	(* 4=zur *)							
	IF hm_zur
		AND NOT temp_end_zur
		AND NOT temp_stoer_zur
		AND NOT temp_stoer_vor_zur
	THEN
		inout_visu.status:=4;									
	END_IF									
	(* 5=ist zur *)							
	IF (temp_end_zur
		OR (NOT inout_visu.para.ueberwachung_zur_aktiv
				AND hm_zur))
		AND NOT temp_end_vor
		AND NOT temp_stoer_zur
		AND NOT temp_stoer_vor_zur
	THEN
		inout_visu.status:=5;									
	END_IF															
	(* 6=Fehler zurück *)								
	IF temp_stoer_zur
	THEN
		inout_visu.status:=6;
	END_IF
	(* 7=Fehler vor zur	*)
	IF temp_stoer_vor_zur
	THEN
		inout_visu.status:=7;
	END_IF

	
(***** Endlagen direkt an die Visu weiter reichen ***********************************************************************************************************)
	out_vor_visu:=in_endlage_vor;
	out_zur_visu:=in_endlage_zur;


(***** IN Start-Befehle Hand und Automatik löschen **********************************************************************************************************)
	inout_ansteuerung.in_auto_vor:=FALSE;
	inout_ansteuerung.in_auto_zur:=FALSE;
	inout_ansteuerung.in_aus := FALSE;
	inout_visu.hand_vor:=FALSE;
	inout_visu.hand_zur:=FALSE;
	hm_timer_reset:=TRUE;

METHOD M_AutoVor : BOOL
VAR_INPUT
	Active		: BOOL;
END_VAR
inout_ansteuerung.in_auto_vor := Active;
IF inout_ansteuerung.out_ist_vor OR NOT Active THEN
	M_AutoVor := TRUE;
END_IF
END_METHOD

METHOD M_AutoZur : BOOL
VAR_INPUT
	Active		: BOOL;
END_VAR
inout_ansteuerung.in_auto_zur := Active;
IF inout_ansteuerung.out_ist_zur OR NOT Active THEN
	M_AutoZur := TRUE;
END_IF
END_METHOD

END_FUNCTION_BLOCK

// ---- 3400_Bohraggregat/Hardware_3400.TcPOU

PROGRAM Hardware_3400
VAR
    // Servos *********************************************************************
	fbX_Achse										: FB_Achse_NC_PTP_Beckhoff; 
	fbY_Achse										: FB_Achse_NC_PTP_Beckhoff; 

    // Frequenzumrichter **********************************************************
	fbBohraggr_Schluessel_ob						: FB_SEW_MOVITRAC_C_CoE;

    // Sensorik *******************************************************************
    fbStillBohraggr_Schluessel_ob          			: FB_Belegt;

    // Ventile ********************************************************************
    fbSchluessel_ob_Bohrhub                			: FB_Ventil_V2;

    // ***** Hilfsmerker***********************************************************
    (*
        Ventile sind über den DUT_Ventil_para vorparametriert
                ueberwachung_vor_aktiv    : BOOL := TRUE;   // 0 = Endlagenüberwachung vor deaktiviert
                ueberwachung_zur_aktiv    : BOOL := TRUE;   // 0 = Endlagenüberwachung zurück deaktiviert
                ausgang_vor_halten        : BOOL := FALSE;  // 1 = Ausgang immer Ein, sonst 0 in Endlage/1 nicht in Endlage
                ausgang_zur_halten        : BOOL := FALSE;  // 1 = Ausgang immer Ein, sonst 0 in Endlage/1 nicht in Endlage
                entprellen_vor_aktiv      : BOOL := TRUE;   // 0 = Endlage sofort überwachen wenn einmal erreicht
                entprellen_zur_aktiv      : BOOL := TRUE;   // 0 = Endlage sofort überwachen wenn einmal erreicht
                ueberwachungszeit_vor     : TIME := T#10S;  // Überwachungszeit in ms (0-30000ms)
                ueberwachungszeit_zur     : TIME := T#10S;  // Überwachungszeit in ms (0-30000ms)
                entprellungszeit_vor      : TIME := T#50MS; // Entprellungszeit in ms (0-10000ms)
                entprellungszeit_zur      : TIME := T#50MS; // Entprellungszeit in ms (0-10000ms)

        falls etwas anderes gewünscht ist, kann man gezielt für das Ventil die Parameter anpassen
        Beispiel:   ***.para.ausgang_vor_halten := TRUE;
                    ***.para.entprellungszeit_vor := T#100MS;
    *)
END_VAR


// Aktionen aufrufen
//_________________________________________________
	A_Sensorik();
	A_Umrichter();
	A_Ventile();
	A_Servo();

ACTION A_Sensorik:
					
// ***** Sensorik entprellen *********************************************************
	//********************************************************************************
fbStillBohraggr_Schluessel_ob	(	in_Sensor:=,
									in_zeit_aus:=T#100MS,
									in_zeit_aus:=T#100MS,
									Q=>);
END_ACTION

ACTION A_Servo:
					
// ***** Servoregler *****************************************************************
	//********************************************************************************
	GVL_3400.X_Achse_steuern.Reglersperre	:= FALSE;
	GVL_3400.X_Achse_steuern.Freigabe 		:= FALSE;
	
	fbX_Achse(
	in_Reglersperre				:= GVL_3400.X_Achse_steuern.Reglersperre, 
	in_Freigabe					:= GVL_3400.X_Achse_steuern.Freigabe,
	in_Reset					:= GVL_Visu_3400.SteuerStatus.reset   
								OR GVL_0000.stoerung_quitt,                      
	in_Hand						:= GVL_Visu_3400.SteuerStatus.hand,              
	in_Auto						:= GVL_Visu_3400.SteuerStatus.auto,                 
	in_Auto_Override			:= GVL_Visu_0000.override,    
	in_Auto_pos					:= , 
	in_PosFenster				:= 0.05, 
	in_Ref_pos					:= 0.0, 
	in_HomingOption				:= , 
	in_EndlageRef				:= , 
	in_DirRef					:= , 
	in_PosEa					:= ,                                       
	out_ist_pos					=> GVL_3400.X_Achse_status.ist_pos, 
	out_in_pos					=> GVL_3400.X_Achse_status.in_pos,   
	out_ziel_pos				=> GVL_3400.X_Achse_status.ziel_pos, 
	out_nicht_ref				=> GVL_3400.X_Achse_status.nicht_ref,      
	out_bremse					=> GVL_3400.X_Achse_status.bremse,           
	out_Achs_Status				=> GVL_3400.X_Achse_status.Achs_Status,  
	inout_NC					:= EAs_3400.ea_X_Achse, 
	inout_service				:= GVL_Visu_3400.X_Achse, 
	inout_Ref_start				:= GVL_3400.X_Achse_steuern.Ref_start, 
	inout_Auto_start			:= GVL_3400.X_Achse_steuern.Auto_start, 
	inout_Auto_stop				:= GVL_3400.X_Achse_steuern.Auto_stop);
	
	GVL_Meldungen.Diagnose_3000.Nr_034	:= fbX_Achse.out_Achs_ErrorID;	
	GVL_Meldungen.Meldungen_3000.Nr_034 := fbX_Achse.out_Achs_Error OR fbX_Achse.out_FB_Error OR fbX_Achse.out_Achs_ErrorID <> 0;		
	GVL_Meldungen.Meldungen_3000.Nr_035 := FALSE;
	GVL_Meldungen.Meldungen_3000.Nr_036 := FALSE;
	//********************************************************************************
					
					
	GVL_3400.Y_Achse_steuern.Reglersperre	:= FALSE;
	GVL_3400.Y_Achse_steuern.Freigabe 		:= FALSE;
	
	fbY_Achse(
	in_Reglersperre				:= GVL_3400.Y_Achse_steuern.Reglersperre, 
	in_Freigabe					:= GVL_3400.Y_Achse_steuern.Freigabe,
	in_Reset					:= GVL_Visu_3400.SteuerStatus.reset   
								OR GVL_0000.stoerung_quitt,                      
	in_Hand						:= GVL_Visu_3400.SteuerStatus.hand,              
	in_Auto						:= GVL_Visu_3400.SteuerStatus.auto,                 
	in_Auto_Override			:= GVL_Visu_0000.override,    
	in_Auto_pos					:= , 
	in_PosFenster				:= 0.05, 
	in_Ref_pos					:= 0.0, 
	in_HomingOption				:= , 
	in_EndlageRef				:= , 
	in_DirRef					:= , 
	in_PosEa					:= ,                                       
	out_ist_pos					=> GVL_3400.Y_Achse_status.ist_pos, 
	out_in_pos					=> GVL_3400.Y_Achse_status.in_pos,   
	out_ziel_pos				=> GVL_3400.Y_Achse_status.ziel_pos, 
	out_nicht_ref				=> GVL_3400.Y_Achse_status.nicht_ref,      
	out_bremse					=> GVL_3400.Y_Achse_status.bremse,           
	out_Achs_Status				=> GVL_3400.Y_Achse_status.Achs_Status,  
	inout_NC					:= EAs_3400.ea_Y_Achse, 
	inout_service				:= GVL_Visu_3400.Y_Achse, 
	inout_Ref_start				:= GVL_3400.Y_Achse_steuern.Ref_start, 
	inout_Auto_start			:= GVL_3400.Y_Achse_steuern.Auto_start, 
	inout_Auto_stop				:= GVL_3400.Y_Achse_steuern.Auto_stop);
	
	GVL_Meldungen.Diagnose_3000.Nr_037	:= fbY_Achse.out_Achs_ErrorID;	
	GVL_Meldungen.Meldungen_3000.Nr_037 := fbY_Achse.out_Achs_Error OR fbY_Achse.out_FB_Error OR fbY_Achse.out_Achs_ErrorID <> 0;		
	GVL_Meldungen.Meldungen_3000.Nr_038 := FALSE;
	GVL_Meldungen.Meldungen_3000.Nr_039 := FALSE;
END_ACTION

ACTION A_Umrichter:
	
// ***** Frequenzumrichter ******************************************************
// ******************************************************************************
				
	GVL_Visu_3400.Bohraggr_Schluessel_ob	.Para.Speed_Hand		:= 0;
	GVL_Visu_3400.Bohraggr_Schluessel_ob	.Para.Beschleunigung 	:= 0;
	GVL_Visu_3400.Bohraggr_Schluessel_ob	.Para.Verzoegerung 		:= 0;
	GVL_Visu_3400.Bohraggr_Schluessel_ob	.Para.Einheit			:= 1;

	fbBohraggr_Schluessel_ob	(	PD_IN	:=EAs_3400.e_Bohraggr_Schluessel_ob	,
			IN_ReglerSperre			:=,
			IN_SteuerStatus			:=GVL_Visu_3400.SteuerStatus,
			IN_Ethercat_Adresse		:=,
			IN_Ethercat_Name		:='',
			IN_QUITTIEREN			:= GVL_0000.stoerung_quitt,
			IN_OVERRIDE				:= GVL_Visu_0000.override,
			PD_OUT					=> EAs_3400.a_Bohraggr_Schluessel_ob	,
			OUT_Stoerung			=> GVL_Meldungen.Meldungen_3000.Nr_007,
			OUT_Fehlernummer		=> GVL_Meldungen.Diagnose_3000.Nr_007,
			OUT_Status				=> GVL_3400.Bohraggr_Schluessel_ob_status,
			inout_visu				:= GVL_Visu_3400.Bohraggr_Schluessel_ob	,
			inout_steuern			:= GVL_3400.Bohraggr_Schluessel_ob_steuern);
	
			GVL_3400.Bohraggr_Schluessel_ob_steuern.vor := FALSE;
			GVL_3400.Bohraggr_Schluessel_ob_steuern.zur := FALSE;
			GVL_3400.Bohraggr_Schluessel_ob_steuern.speed := 0;
END_ACTION

ACTION A_Ventile:
	
// ***** Ventile *********************************************************************
	//********************************************************************************	
	
	GVL_Visu_3400.Schluessel_ob_Bohrhub.para.ausgang_vor_halten:=TRUE;	
	GVL_Visu_3400.Schluessel_ob_Bohrhub.para.ausgang_zur_halten:=TRUE;	
	GVL_Visu_3400.Schluessel_ob_Bohrhub.para.ueberwachung_vor_aktiv:=TRUE;	
	GVL_Visu_3400.Schluessel_ob_Bohrhub.para.ueberwachung_zur_aktiv:=TRUE;	
	GVL_Visu_3400.Schluessel_ob_Bohrhub.para.entprellungszeit_vor:=T#50S;	
	GVL_Visu_3400.Schluessel_ob_Bohrhub.para.entprellungszeit_zur:=T#50MS;	
	fbSchluessel_ob_Bohrhub (	in_endlage_vor:= EAs_3400.e_FR_3400_Druecker_Schluesselloch_oben_Bohraggregat_7_Bohrhub_ist_oben,
								in_endlage_zur:= EAs_3400.e_FR_3400_Druecker_Schluesselloch_oben_Bohraggregat_7_Bohrhub_ist_unten,
								in_hand:=GVL_Visu_3400.SteuerStatus.hand,
								in_auto:=GVL_Visu_3400.SteuerStatus.auto,
								in_quit:=GVL_Visu_3400.SteuerStatus.reset 
								OR GVL_0000.stoerung_quitt,
								out_vor=>EAs_3400.a_FR_3400_Druecker_Schluesselloch_oben_Bohraggregat_7_Bohrhub_heben,
								out_zur=>EAs_3400.a_FR_3400_Druecker_Schluesselloch_oben_Bohraggregat_7_Bohrhub_senken,
								out_stoerung_vor=> GVL_Meldungen.Meldungen_3000.Nr_070,
								out_stoerung_zur=> GVL_Meldungen.Meldungen_3000.Nr_071,
								out_stoerung_vorzur=> GVL_Meldungen.Meldungen_3000.Nr_072,
								inout_ansteuerung:=GVL_3400.Schluessel_ob_Bohrhub ,
								inout_visu:=GVL_Visu_3400.Schluessel_ob_Bohrhub );
END_ACTION

END_PROGRAM

// ---- 3510_Transport/Ablauf_3510.TcPOU

PROGRAM Ablauf_3510
VAR
    // TODO: lokale Variablen fuer den Ablauf deklarieren
END_VAR


// TODO: Hauptprogramm-Code fuer Ablauf hier einfuegen


METHOD M_VisuKomm : BOOL
VAR_INPUT
    Nr          : INT;
END_VAR
VAR_IN_OUT
    anVisu      : INT;
    vonVisu     : INT;
END_VAR

VAR_INST
    result                  : INT;
    ton_DatenUngueltig      : TON;
    ton_DatenTimeout        : TON;
    sc                      : INT;
END_VAR

// Schnistelle zur VISU Kommunikation
// Starttrigger belegen als Antwort wird auf die 5= gut oder 9=schlecht gewartet.
// Kommunikationstimeout nach 5 Sekunden und wird automatisch wieder neugestartet

ton_DatenTimeout(IN:= anVisu <> 0 AND vonVisu = 0, PT:=T#3S);
ton_DatenUngueltig(IN:= sc = 20, PT:=T#500MS);

CASE sc OF
    0:  // Anfrage starten und auf Antwort warten
        anVisu := Nr;
        result := 0;
        IF vonVisu <> 0 THEN
            IF (vonVisu MOD Nr) = 5 THEN
                sc := 10;
            ELSIF (vonVisu MOD Nr) = 9 THEN
                sc := 20;
            END_IF
        ELSIF ton_DatenTimeout.Q THEN
            sc := 20;
        END_IF

    10: // Antwort 5 erhalten
        anVisu := 0;
        IF vonVisu = 0 THEN
            M_VisuKomm := TRUE;
            result := 1;
            sc := 0;
        END_IF

    20: // Timeout, 1 Sekunde warten und erneut antriggern
        IF ton_DatenUngueltig.Q THEN
            anVisu := 0;
            IF vonVisu = 0 THEN
                result := -1;
                sc := 0;
            END_IF
        END_IF

END_CASE
END_METHOD


METHOD M_VisuKommInt : INT
VAR_INPUT
    Nr          : INT;
END_VAR
VAR_IN_OUT
    anVisu      : INT;
    vonVisu     : INT;
END_VAR

VAR_INST
    result                  : INT;
    ton_DatenUngueltig      : TON;
    ton_DatenTimeout        : TON;
    sc                      : INT;
END_VAR

// Schnistelle zur VISU Kommunikation
// Starttrigger belegen als Antwort wird auf die 5= gut oder 9=schlecht gewartet.
// Kommunikationstimeout nach 5 Sekunden und wird automatisch wieder neugestartet

ton_DatenTimeout(IN:= anVisu <> 0 AND vonVisu = 0, PT:=T#3S);
ton_DatenUngueltig(IN:= anVisu = 0 AND vonVisu = 0, PT:=T#500MS);

CASE sc OF
    0:  // Anfrage starten und auf Antwort warten
        anVisu := Nr;
        result := 0;
        IF vonVisu <> 0 THEN
            IF (vonVisu MOD Nr) = 5 THEN
                sc := 10;
            ELSIF (vonVisu MOD Nr) = 9 THEN
                sc := 15;
            END_IF
        ELSIF ton_DatenTimeout.Q THEN
            sc := 20;
        END_IF

    10: // Antwort 5 erhalten (OK)
        anVisu := 0;
        IF vonVisu = 0 THEN
            M_VisuKommInt := 1;
            result := 1;
            sc := 0;
        END_IF

    15: // Antwort 9 erhalten (Fehler)
        anVisu := 0;
        IF vonVisu = 0 THEN
            M_VisuKommInt := -1;
            result := 1;
            sc := 0;
        END_IF

    20: // Timeout, 1 Sekunde warten und erneut antriggern
        anVisu := 0;
        IF vonVisu = 0 THEN
            result := -1;
            IF ton_DatenUngueltig.Q THEN
                sc := 0;
            END_IF
        END_IF

END_CASE
END_METHOD

END_PROGRAM

// ---- 3510_Transport/Hardware_3510.TcPOU

PROGRAM Hardware_3510
VAR
    // Servos *********************************************************************
    //fbAchse                   	 				: FB_Achse_NC_PTP_V4_1; 

    // Frequenzumrichter **********************************************************
	fbTrans_Schlossseite							: FB_SEW_MOVITRAC_C_CoE;

    // Sensorik *******************************************************************
    fbLangsam          								: FB_Belegt;
    fbStopp         								: FB_Belegt;
    fbLaengsSchlossseite_Ref						: FB_Belegt;

    // Ventile ********************************************************************
    fbLaengsanschl                					: FB_Ventil_V2;
    fbSchienenklemm               					: FB_Ventil_V2;

    // ***** Hilfsmerker***********************************************************
    (*
        Ventile sind über den DUT_Ventil_para vorparametriert
                ueberwachung_vor_aktiv    : BOOL := TRUE;   // 0 = Endlagenüberwachung vor deaktiviert
                ueberwachung_zur_aktiv    : BOOL := TRUE;   // 0 = Endlagenüberwachung zurück deaktiviert
                ausgang_vor_halten        : BOOL := FALSE;  // 1 = Ausgang immer Ein, sonst 0 in Endlage/1 nicht in Endlage
                ausgang_zur_halten        : BOOL := FALSE;  // 1 = Ausgang immer Ein, sonst 0 in Endlage/1 nicht in Endlage
                entprellen_vor_aktiv      : BOOL := TRUE;   // 0 = Endlage sofort überwachen wenn einmal erreicht
                entprellen_zur_aktiv      : BOOL := TRUE;   // 0 = Endlage sofort überwachen wenn einmal erreicht
                ueberwachungszeit_vor     : TIME := T#10S;  // Überwachungszeit in ms (0-30000ms)
                ueberwachungszeit_zur     : TIME := T#10S;  // Überwachungszeit in ms (0-30000ms)
                entprellungszeit_vor      : TIME := T#50MS; // Entprellungszeit in ms (0-10000ms)
                entprellungszeit_zur      : TIME := T#50MS; // Entprellungszeit in ms (0-10000ms)

        falls etwas anderes gewünscht ist, kann man gezielt für das Ventil die Parameter anpassen
        Beispiel:   ***.para.ausgang_vor_halten := TRUE;
                    ***.para.entprellungszeit_vor := T#100MS;
    *)
END_VAR


// Aktionen aufrufen
//_________________________________________________
	A_Sensorik();
	A_Umrichter();
	A_Ventile();
	A_Servo();

ACTION A_Sensorik:
					
// ***** Sensorik entprellen *********************************************************
	//********************************************************************************
fbLangsam						(	in_Sensor:=,
									in_zeit_aus:=T#100MS,
									in_zeit_aus:=T#100MS,
									Q=>);
									
fbStopp							(	in_Sensor:=,
									in_zeit_aus:=T#100MS,
									in_zeit_aus:=T#100MS,
									Q=>);
									
fbLaengsSchlossseite_Ref		(	in_Sensor:=,
									in_zeit_aus:=T#100MS,
									in_zeit_aus:=T#100MS,
									Q=>);
END_ACTION

ACTION A_Servo:

END_ACTION

ACTION A_Umrichter:

// ***** Frequenzumrichter ******************************************************
// ******************************************************************************
				
	GVL_Visu_3510.Trans_Schlossseite	.Para.Speed_Hand		:= 0;
	GVL_Visu_3510.Trans_Schlossseite	.Para.Beschleunigung 	:= 0;
	GVL_Visu_3510.Trans_Schlossseite	.Para.Verzoegerung 		:= 0;
	GVL_Visu_3510.Trans_Schlossseite	.Para.Einheit			:= 1;

	fbTrans_Schlossseite	(	PD_IN	:=EAs_3510.e_Trans_Schlossseite	,
			IN_ReglerSperre			:=,
			IN_SteuerStatus			:=GVL_Visu_3510.SteuerStatus,
			IN_Ethercat_Adresse		:=,
			IN_Ethercat_Name		:='',
			IN_QUITTIEREN			:= GVL_0000.stoerung_quitt,
			IN_OVERRIDE				:= GVL_Visu_0000.override,
			PD_OUT					=> EAs_3510.a_Trans_Schlossseite	,
			OUT_Stoerung			=> GVL_Meldungen.Meldungen_3000.Nr_008,
			OUT_Fehlernummer		=> GVL_Meldungen.Diagnose_3000.Nr_008,
			OUT_Status				=> GVL_3510.Trans_Schlossseite_status,
			inout_visu				:= GVL_Visu_3510.Trans_Schlossseite	,
			inout_steuern			:= GVL_3510.Trans_Schlossseite_steuern);
	
			GVL_3510.Trans_Schlossseite_steuern.vor := FALSE;
			GVL_3510.Trans_Schlossseite_steuern.zur := FALSE;
			GVL_3510.Trans_Schlossseite_steuern.speed := 0;
END_ACTION

ACTION A_Ventile:
	
// ***** Ventile *********************************************************************
	//********************************************************************************	
	
	GVL_Visu_3510.Laengsanschl.para.ausgang_vor_halten:=TRUE;	
	GVL_Visu_3510.Laengsanschl.para.ausgang_zur_halten:=TRUE;	
	GVL_Visu_3510.Laengsanschl.para.ueberwachung_vor_aktiv:=TRUE;	
	GVL_Visu_3510.Laengsanschl.para.ueberwachung_zur_aktiv:=TRUE;	
	GVL_Visu_3510.Laengsanschl.para.entprellungszeit_vor:=T#50S;	
	GVL_Visu_3510.Laengsanschl.para.entprellungszeit_zur:=T#50MS;	
	fbLaengsanschl (		in_endlage_vor:= ,
							in_endlage_zur:= ,
							in_hand:=GVL_Visu_3510.SteuerStatus.hand,
							in_auto:=GVL_Visu_3510.SteuerStatus.auto,
							in_quit:=GVL_Visu_3510.SteuerStatus.reset 
							OR GVL_0000.stoerung_quitt,
							out_vor=>,
							out_zur=>,
							out_stoerung_vor=> GVL_Meldungen.Meldungen_3000.Nr_073,
							out_stoerung_zur=> GVL_Meldungen.Meldungen_3000.Nr_074,
							out_stoerung_vorzur=> GVL_Meldungen.Meldungen_3000.Nr_075,
							inout_ansteuerung:=GVL_3510.Laengsanschl ,
							inout_visu:=GVL_Visu_3510.Laengsanschl );
								
	
	GVL_Visu_3510.Schienenklemm.para.ausgang_vor_halten:=TRUE;	
	GVL_Visu_3510.Schienenklemm.para.ausgang_zur_halten:=TRUE;	
	GVL_Visu_3510.Schienenklemm.para.ueberwachung_vor_aktiv:=TRUE;	
	GVL_Visu_3510.Schienenklemm.para.ueberwachung_zur_aktiv:=TRUE;	
	GVL_Visu_3510.Schienenklemm.para.entprellungszeit_vor:=T#500MS;	
	GVL_Visu_3510.Schienenklemm.para.entprellungszeit_zur:=T#500MS;	
	fbSchienenklemm(			in_endlage_vor:= EAs_3510.a_FR_3510_Transport_Schlossseite_X_Achse_Laengsanschlag_Schienenklemmung_klemmen, 
								in_endlage_zur:= NOT EAs_3510.a_FR_3510_Transport_Schlossseite_X_Achse_Laengsanschlag_Schienenklemmung_klemmen,
								in_hand:=GVL_Visu_3510.SteuerStatus.hand,
								in_auto:=GVL_Visu_3510.SteuerStatus.auto,
								in_quit:=GVL_Visu_3510.SteuerStatus.reset 
								OR GVL_0000.stoerung_quitt,
								out_vor=>EAs_3510.a_FR_3510_Transport_Schlossseite_X_Achse_Laengsanschlag_Schienenklemmung_klemmen,
								out_zur=>,
								out_stoerung_vor=> GVL_Meldungen.Meldungen_3000.Nr_088,
								out_stoerung_zur=> GVL_Meldungen.Meldungen_3000.Nr_089,
								out_stoerung_vorzur=> GVL_Meldungen.Meldungen_3000.Nr_090,
								inout_ansteuerung:=GVL_3510.Schienenklemm,
								inout_visu:=GVL_Visu_3510.Schienenklemm);
END_ACTION

END_PROGRAM

// ---- 3520_Transport/Ablauf_3520.TcPOU

PROGRAM Ablauf_3520
VAR
    // TODO: lokale Variablen fuer den Ablauf deklarieren
END_VAR


// TODO: Hauptprogramm-Code fuer Ablauf hier einfuegen


METHOD M_VisuKomm : BOOL
VAR_INPUT
    Nr          : INT;
END_VAR
VAR_IN_OUT
    anVisu      : INT;
    vonVisu     : INT;
END_VAR

VAR_INST
    result                  : INT;
    ton_DatenUngueltig      : TON;
    ton_DatenTimeout        : TON;
    sc                      : INT;
END_VAR

// Schnistelle zur VISU Kommunikation
// Starttrigger belegen als Antwort wird auf die 5= gut oder 9=schlecht gewartet.
// Kommunikationstimeout nach 5 Sekunden und wird automatisch wieder neugestartet

ton_DatenTimeout(IN:= anVisu <> 0 AND vonVisu = 0, PT:=T#3S);
ton_DatenUngueltig(IN:= sc = 20, PT:=T#500MS);

CASE sc OF
    0:  // Anfrage starten und auf Antwort warten
        anVisu := Nr;
        result := 0;
        IF vonVisu <> 0 THEN
            IF (vonVisu MOD Nr) = 5 THEN
                sc := 10;
            ELSIF (vonVisu MOD Nr) = 9 THEN
                sc := 20;
            END_IF
        ELSIF ton_DatenTimeout.Q THEN
            sc := 20;
        END_IF

    10: // Antwort 5 erhalten
        anVisu := 0;
        IF vonVisu = 0 THEN
            M_VisuKomm := TRUE;
            result := 1;
            sc := 0;
        END_IF

    20: // Timeout, 1 Sekunde warten und erneut antriggern
        IF ton_DatenUngueltig.Q THEN
            anVisu := 0;
            IF vonVisu = 0 THEN
                result := -1;
                sc := 0;
            END_IF
        END_IF

END_CASE
END_METHOD


METHOD M_VisuKommInt : INT
VAR_INPUT
    Nr          : INT;
END_VAR
VAR_IN_OUT
    anVisu      : INT;
    vonVisu     : INT;
END_VAR

VAR_INST
    result                  : INT;
    ton_DatenUngueltig      : TON;
    ton_DatenTimeout        : TON;
    sc                      : INT;
END_VAR

// Schnistelle zur VISU Kommunikation
// Starttrigger belegen als Antwort wird auf die 5= gut oder 9=schlecht gewartet.
// Kommunikationstimeout nach 5 Sekunden und wird automatisch wieder neugestartet

ton_DatenTimeout(IN:= anVisu <> 0 AND vonVisu = 0, PT:=T#3S);
ton_DatenUngueltig(IN:= anVisu = 0 AND vonVisu = 0, PT:=T#500MS);

CASE sc OF
    0:  // Anfrage starten und auf Antwort warten
        anVisu := Nr;
        result := 0;
        IF vonVisu <> 0 THEN
            IF (vonVisu MOD Nr) = 5 THEN
                sc := 10;
            ELSIF (vonVisu MOD Nr) = 9 THEN
                sc := 15;
            END_IF
        ELSIF ton_DatenTimeout.Q THEN
            sc := 20;
        END_IF

    10: // Antwort 5 erhalten (OK)
        anVisu := 0;
        IF vonVisu = 0 THEN
            M_VisuKommInt := 1;
            result := 1;
            sc := 0;
        END_IF

    15: // Antwort 9 erhalten (Fehler)
        anVisu := 0;
        IF vonVisu = 0 THEN
            M_VisuKommInt := -1;
            result := 1;
            sc := 0;
        END_IF

    20: // Timeout, 1 Sekunde warten und erneut antriggern
        anVisu := 0;
        IF vonVisu = 0 THEN
            result := -1;
            IF ton_DatenUngueltig.Q THEN
                sc := 0;
            END_IF
        END_IF

END_CASE
END_METHOD

END_PROGRAM

// ---- 3530_Niederhalter/Ablauf_3530.TcPOU

PROGRAM Ablauf_3530
VAR
    // TODO: lokale Variablen fuer den Ablauf deklarieren
END_VAR


// TODO: Hauptprogramm-Code fuer Ablauf hier einfuegen


METHOD M_VisuKomm : BOOL
VAR_INPUT
    Nr          : INT;
END_VAR
VAR_IN_OUT
    anVisu      : INT;
    vonVisu     : INT;
END_VAR

VAR_INST
    result                  : INT;
    ton_DatenUngueltig      : TON;
    ton_DatenTimeout        : TON;
    sc                      : INT;
END_VAR

// Schnistelle zur VISU Kommunikation
// Starttrigger belegen als Antwort wird auf die 5= gut oder 9=schlecht gewartet.
// Kommunikationstimeout nach 5 Sekunden und wird automatisch wieder neugestartet

ton_DatenTimeout(IN:= anVisu <> 0 AND vonVisu = 0, PT:=T#3S);
ton_DatenUngueltig(IN:= sc = 20, PT:=T#500MS);

CASE sc OF
    0:  // Anfrage starten und auf Antwort warten
        anVisu := Nr;
        result := 0;
        IF vonVisu <> 0 THEN
            IF (vonVisu MOD Nr) = 5 THEN
                sc := 10;
            ELSIF (vonVisu MOD Nr) = 9 THEN
                sc := 20;
            END_IF
        ELSIF ton_DatenTimeout.Q THEN
            sc := 20;
        END_IF

    10: // Antwort 5 erhalten
        anVisu := 0;
        IF vonVisu = 0 THEN
            M_VisuKomm := TRUE;
            result := 1;
            sc := 0;
        END_IF

    20: // Timeout, 1 Sekunde warten und erneut antriggern
        IF ton_DatenUngueltig.Q THEN
            anVisu := 0;
            IF vonVisu = 0 THEN
                result := -1;
                sc := 0;
            END_IF
        END_IF

END_CASE
END_METHOD


METHOD M_VisuKommInt : INT
VAR_INPUT
    Nr          : INT;
END_VAR
VAR_IN_OUT
    anVisu      : INT;
    vonVisu     : INT;
END_VAR

VAR_INST
    result                  : INT;
    ton_DatenUngueltig      : TON;
    ton_DatenTimeout        : TON;
    sc                      : INT;
END_VAR

// Schnistelle zur VISU Kommunikation
// Starttrigger belegen als Antwort wird auf die 5= gut oder 9=schlecht gewartet.
// Kommunikationstimeout nach 5 Sekunden und wird automatisch wieder neugestartet

ton_DatenTimeout(IN:= anVisu <> 0 AND vonVisu = 0, PT:=T#3S);
ton_DatenUngueltig(IN:= anVisu = 0 AND vonVisu = 0, PT:=T#500MS);

CASE sc OF
    0:  // Anfrage starten und auf Antwort warten
        anVisu := Nr;
        result := 0;
        IF vonVisu <> 0 THEN
            IF (vonVisu MOD Nr) = 5 THEN
                sc := 10;
            ELSIF (vonVisu MOD Nr) = 9 THEN
                sc := 15;
            END_IF
        ELSIF ton_DatenTimeout.Q THEN
            sc := 20;
        END_IF

    10: // Antwort 5 erhalten (OK)
        anVisu := 0;
        IF vonVisu = 0 THEN
            M_VisuKommInt := 1;
            result := 1;
            sc := 0;
        END_IF

    15: // Antwort 9 erhalten (Fehler)
        anVisu := 0;
        IF vonVisu = 0 THEN
            M_VisuKommInt := -1;
            result := 1;
            sc := 0;
        END_IF

    20: // Timeout, 1 Sekunde warten und erneut antriggern
        anVisu := 0;
        IF vonVisu = 0 THEN
            result := -1;
            IF ton_DatenUngueltig.Q THEN
                sc := 0;
            END_IF
        END_IF

END_CASE
END_METHOD

END_PROGRAM

// ---- 3540_Niederhalter/Ablauf_3540.TcPOU

PROGRAM Ablauf_3540
VAR
    // TODO: lokale Variablen fuer den Ablauf deklarieren
END_VAR


// TODO: Hauptprogramm-Code fuer Ablauf hier einfuegen


METHOD M_VisuKomm : BOOL
VAR_INPUT
    Nr          : INT;
END_VAR
VAR_IN_OUT
    anVisu      : INT;
    vonVisu     : INT;
END_VAR

VAR_INST
    result                  : INT;
    ton_DatenUngueltig      : TON;
    ton_DatenTimeout        : TON;
    sc                      : INT;
END_VAR

// Schnistelle zur VISU Kommunikation
// Starttrigger belegen als Antwort wird auf die 5= gut oder 9=schlecht gewartet.
// Kommunikationstimeout nach 5 Sekunden und wird automatisch wieder neugestartet

ton_DatenTimeout(IN:= anVisu <> 0 AND vonVisu = 0, PT:=T#3S);
ton_DatenUngueltig(IN:= sc = 20, PT:=T#500MS);

CASE sc OF
    0:  // Anfrage starten und auf Antwort warten
        anVisu := Nr;
        result := 0;
        IF vonVisu <> 0 THEN
            IF (vonVisu MOD Nr) = 5 THEN
                sc := 10;
            ELSIF (vonVisu MOD Nr) = 9 THEN
                sc := 20;
            END_IF
        ELSIF ton_DatenTimeout.Q THEN
            sc := 20;
        END_IF

    10: // Antwort 5 erhalten
        anVisu := 0;
        IF vonVisu = 0 THEN
            M_VisuKomm := TRUE;
            result := 1;
            sc := 0;
        END_IF

    20: // Timeout, 1 Sekunde warten und erneut antriggern
        IF ton_DatenUngueltig.Q THEN
            anVisu := 0;
            IF vonVisu = 0 THEN
                result := -1;
                sc := 0;
            END_IF
        END_IF

END_CASE
END_METHOD


METHOD M_VisuKommInt : INT
VAR_INPUT
    Nr          : INT;
END_VAR
VAR_IN_OUT
    anVisu      : INT;
    vonVisu     : INT;
END_VAR

VAR_INST
    result                  : INT;
    ton_DatenUngueltig      : TON;
    ton_DatenTimeout        : TON;
    sc                      : INT;
END_VAR

// Schnistelle zur VISU Kommunikation
// Starttrigger belegen als Antwort wird auf die 5= gut oder 9=schlecht gewartet.
// Kommunikationstimeout nach 5 Sekunden und wird automatisch wieder neugestartet

ton_DatenTimeout(IN:= anVisu <> 0 AND vonVisu = 0, PT:=T#3S);
ton_DatenUngueltig(IN:= anVisu = 0 AND vonVisu = 0, PT:=T#500MS);

CASE sc OF
    0:  // Anfrage starten und auf Antwort warten
        anVisu := Nr;
        result := 0;
        IF vonVisu <> 0 THEN
            IF (vonVisu MOD Nr) = 5 THEN
                sc := 10;
            ELSIF (vonVisu MOD Nr) = 9 THEN
                sc := 15;
            END_IF
        ELSIF ton_DatenTimeout.Q THEN
            sc := 20;
        END_IF

    10: // Antwort 5 erhalten (OK)
        anVisu := 0;
        IF vonVisu = 0 THEN
            M_VisuKommInt := 1;
            result := 1;
            sc := 0;
        END_IF

    15: // Antwort 9 erhalten (Fehler)
        anVisu := 0;
        IF vonVisu = 0 THEN
            M_VisuKommInt := -1;
            result := 1;
            sc := 0;
        END_IF

    20: // Timeout, 1 Sekunde warten und erneut antriggern
        anVisu := 0;
        IF vonVisu = 0 THEN
            result := -1;
            IF ton_DatenUngueltig.Q THEN
                sc := 0;
            END_IF
        END_IF

END_CASE
END_METHOD

END_PROGRAM

// ---- 3540_Niederhalter/Hardware_3540.TcPOU

PROGRAM Hardware_3540
VAR
    // Servos *********************************************************************
	fbY_Achse										: FB_Achse_NC_PTP_Beckhoff; 

    // Frequenzumrichter **********************************************************
    //fbTransport                					: FB_SEW_MOVITRAC_C_CoE;

    // Sensorik *******************************************************************
    //fbSensor                   					: FB_Belegt;

    // Ventile ********************************************************************
    fbNiederhalter                					: FB_Ventil_V2;

    // ***** Hilfsmerker***********************************************************
    (*
        Ventile sind über den DUT_Ventil_para vorparametriert
                ueberwachung_vor_aktiv    : BOOL := TRUE;   // 0 = Endlagenüberwachung vor deaktiviert
                ueberwachung_zur_aktiv    : BOOL := TRUE;   // 0 = Endlagenüberwachung zurück deaktiviert
                ausgang_vor_halten        : BOOL := FALSE;  // 1 = Ausgang immer Ein, sonst 0 in Endlage/1 nicht in Endlage
                ausgang_zur_halten        : BOOL := FALSE;  // 1 = Ausgang immer Ein, sonst 0 in Endlage/1 nicht in Endlage
                entprellen_vor_aktiv      : BOOL := TRUE;   // 0 = Endlage sofort überwachen wenn einmal erreicht
                entprellen_zur_aktiv      : BOOL := TRUE;   // 0 = Endlage sofort überwachen wenn einmal erreicht
                ueberwachungszeit_vor     : TIME := T#10S;  // Überwachungszeit in ms (0-30000ms)
                ueberwachungszeit_zur     : TIME := T#10S;  // Überwachungszeit in ms (0-30000ms)
                entprellungszeit_vor      : TIME := T#50MS; // Entprellungszeit in ms (0-10000ms)
                entprellungszeit_zur      : TIME := T#50MS; // Entprellungszeit in ms (0-10000ms)

        falls etwas anderes gewünscht ist, kann man gezielt für das Ventil die Parameter anpassen
        Beispiel:   ***.para.ausgang_vor_halten := TRUE;
                    ***.para.entprellungszeit_vor := T#100MS;
    *)
END_VAR


// Aktionen aufrufen
//_________________________________________________
	A_Sensorik();
	A_Umrichter();
	A_Ventile();
	A_Servo();

ACTION A_Sensorik:

END_ACTION

ACTION A_Servo:
					
// ***** Servoregler *****************************************************************
	//********************************************************************************
								
	GVL_3540.Y_Achse_steuern.Reglersperre	:= FALSE;
	GVL_3540.Y_Achse_steuern.Freigabe 		:= FALSE;
	
	fbY_Achse(
	in_Reglersperre				:= GVL_3540.Y_Achse_steuern.Reglersperre, 
	in_Freigabe					:= GVL_3540.Y_Achse_steuern.Freigabe,
	in_Reset					:= GVL_Visu_3540.SteuerStatus.reset   
								OR GVL_0000.stoerung_quitt,                      
	in_Hand						:= GVL_Visu_3540.SteuerStatus.hand,              
	in_Auto						:= GVL_Visu_3540.SteuerStatus.auto,                 
	in_Auto_Override			:= GVL_Visu_0000.override,    
	in_Auto_pos					:= , 
	in_PosFenster				:= 0.05, 
	in_Ref_pos					:= 0.0, 
	in_HomingOption				:= , 
	in_EndlageRef				:= , 
	in_DirRef					:= , 
	in_PosEa					:= ,                                       
	out_ist_pos					=> GVL_3540.Y_Achse_status.ist_pos, 
	out_in_pos					=> GVL_3540.Y_Achse_status.in_pos,   
	out_ziel_pos				=> GVL_3540.Y_Achse_status.ziel_pos, 
	out_nicht_ref				=> GVL_3540.Y_Achse_status.nicht_ref,      
	out_bremse					=> GVL_3540.Y_Achse_status.bremse,           
	out_Achs_Status				=> GVL_3540.Y_Achse_status.Achs_Status,  
	inout_NC					:= EAs_3540.ea_Y_Achse, 
	inout_service				:= GVL_Visu_3540.Y_Achse, 
	inout_Ref_start				:= GVL_3540.Y_Achse_steuern.Ref_start, 
	inout_Auto_start			:= GVL_3540.Y_Achse_steuern.Auto_start, 
	inout_Auto_stop				:= GVL_3540.Y_Achse_steuern.Auto_stop);
	
	GVL_Meldungen.Diagnose_3000.Nr_043	:= fbY_Achse.out_Achs_ErrorID;	
	GVL_Meldungen.Meldungen_3000.Nr_043 := fbY_Achse.out_Achs_Error OR fbY_Achse.out_FB_Error OR fbY_Achse.out_Achs_ErrorID <> 0;		
	GVL_Meldungen.Meldungen_3000.Nr_044 := FALSE;
	GVL_Meldungen.Meldungen_3000.Nr_045 := FALSE;
END_ACTION

ACTION A_Umrichter:

END_ACTION

ACTION A_Ventile:
	
// ***** Ventile *********************************************************************
	//********************************************************************************	
	
	GVL_Visu_3540.Niederhalter.para.ausgang_vor_halten:=TRUE;	
	GVL_Visu_3540.Niederhalter.para.ausgang_zur_halten:=TRUE;	
	GVL_Visu_3540.Niederhalter.para.ueberwachung_vor_aktiv:=TRUE;	
	GVL_Visu_3540.Niederhalter.para.ueberwachung_zur_aktiv:=TRUE;	
	GVL_Visu_3540.Niederhalter.para.entprellungszeit_vor:=T#50S;	
	GVL_Visu_3540.Niederhalter.para.entprellungszeit_zur:=T#50MS;	
	fbNiederhalter (		in_endlage_vor:= EAs_3540.e_FR_3540_Niederhalter_Bandseite_Niederhalter_Einlauf_ist_oben
							AND EAs_3540.e_FR_3540_Niederhalter_Bandseite_Niederhalter_Auslauf_ist_oben,
							in_endlage_zur:= EAs_3540.e_FR_3540_Niederhalter_Bandseite_Niederhalter_Einlauf_ist_unten
							AND EAs_3540.e_FR_3540_Niederhalter_Bandseite_Niederhalter_Auslauf_ist_unten,
							in_hand:=GVL_Visu_3540.SteuerStatus.hand,
							in_auto:=GVL_Visu_3540.SteuerStatus.auto,
							in_quit:=GVL_Visu_3540.SteuerStatus.reset 
							OR GVL_0000.stoerung_quitt,
							out_vor=>EAs_3540.a_FR_3540_Niederhalter_Bandseite_Niederhalter_heben,
							out_zur=>EAs_3540.a_FR_3540_Niederhalter_Bandseite_Niederhalter_senken,
							out_stoerung_vor=> GVL_Meldungen.Meldungen_3000.Nr_079,
							out_stoerung_zur=> GVL_Meldungen.Meldungen_3000.Nr_080,
							out_stoerung_vorzur=> GVL_Meldungen.Meldungen_3000.Nr_081,
							inout_ansteuerung:=GVL_3540.Niederhalter ,
							inout_visu:=GVL_Visu_3540.Niederhalter );
END_ACTION

END_PROGRAM

// ---- SRT_Allgemein/0010_Bausteine_mitDuts/POUs/FB_Achs_Freigabe.TcPOU
FUNCTION_BLOCK FB_Achs_Freigabe
VAR_INPUT
	in_service 		: DUT_Achse_Service;
	in_steuern 		: DUT_Achse_Steuern;
	in_status  		: DUT_Achse_Status;
	in_steuerstatus : DUT_Visu_SteuerStatus;
	in_Einrichtbetrieb : BOOL;
	in_Bedingung_negativ : BOOL;
	in_Bedingung_positiv : BOOL;
	in_min_pos	: REAL;
	in_max_pos	: REAL;
END_VAR
VAR_OUTPUT
	out_Freigabe : BOOL;
	out_Meldung_Einrichtbetrieb : BOOL;
END_VAR
VAR_IN_OUT
	inout_Stoerung : BOOL; // Störung keine Freigabe wenn Startbefehl aktiv (Handbetrieb)
END_VAR
VAR
	Sollrichtung : INT; // 1= positiv, 2= negativ
	Zielposition : REAL;
END_VAR

// FB zur Erzeugng von Achsfreigaben
// Freigabe abhängig von Sollrichtung und jeweiliger Bedingung

Sollrichtung_pruefen();

// Freigabe positiv
IF Sollrichtung = 1
	AND (in_Bedingung_positiv	
		OR (in_steuerstatus.hand
			AND in_service.betriebsart = 1
			AND in_service.minus_stop))
	AND in_status.ist_pos <= in_max_pos	
	AND (Zielposition <= in_max_pos	
		OR (in_steuerstatus.hand
			AND in_service.betriebsart = 1))
THEN
	out_Freigabe := TRUE;
	
// Freigabe negativ
ELSIF Sollrichtung = 2
	AND (in_Bedingung_negativ
		OR (in_steuerstatus.hand
			AND in_service.betriebsart = 1
			AND in_service.minus_stop))
	AND in_status.ist_pos >= in_min_pos
	AND (Zielposition >= in_min_pos
		OR (in_steuerstatus.hand
			AND in_service.betriebsart = 1))
THEN	
	out_Freigabe := TRUE;

// Keine Richtung - Soll gleich ist	
ELSIF Sollrichtung = 0
THEN
	out_Freigabe := TRUE;
	
// Keine Freigabe
ELSE
	out_Freigabe := FALSE;
END_IF

// Störmeldung erzeugen
IF (NOT out_Freigabe
	AND in_steuerstatus.hand
	AND ((in_service.betriebsart = 1	// Tippen
		AND (in_service.minus_stop
			OR in_service.plus_start))
		OR (in_service.betriebsart = 2 	// Positionieren
			AND in_service.plus_start))	)	
	//OR NOT in_Bedingung_negativ
	//OR NOT in_Bedingung_positiv	
THEN
	inout_Stoerung := TRUE;
END_IF

// Einrichtbetrieb
IF in_Einrichtbetrieb
	AND in_steuerstatus.hand
THEN
	inout_Stoerung 	:= FALSE;
	out_Freigabe	:= TRUE;
END_IF

ACTION Sollrichtung_pruefen:
// Zielposition ermitteln
IF in_Status.Achs_Status.Moving
THEN
	Zielposition := in_status.ziel_pos;
ELSIF in_steuerstatus.auto
	AND in_steuern.Auto_start
THEN
	Zielposition := in_steuern.Auto_pos;
ELSIF in_steuerstatus.hand
	AND in_service.betriebsart = 2				
			AND in_service.plus_start
THEN
	Zielposition := in_service.sollpos_hand;	
END_IF	

// Sollrichtung Automatik *************************************************************************
IF in_SteuerStatus.auto
THEN
	IF Zielposition < in_status.ist_pos
	THEN
		Sollrichtung := 2;
	ELSIF Zielposition > in_status.ist_pos
	THEN 
		Sollrichtung := 1;
	ELSE
		Sollrichtung := 0;
	END_IF
	
// Sollrichtung Hand *****************************************************************************	
ELSIF in_SteuerStatus.hand
THEN
	// Tippen
	IF in_service.betriebsart = 1
	THEN
		IF in_service.minus_stop
		THEN
			Sollrichtung := 2;
		ELSIF in_service.plus_start 
		THEN
			Sollrichtung := 1;
		ELSE
			Sollrichtung := 0;
		END_IF
		
	// Positionieren
	ELSIF in_service.betriebsart = 2
	THEN
		IF Zielposition < in_status.ist_pos
		THEN		
			Sollrichtung := 2;
			
		ELSIF Zielposition > in_status.ist_pos
		THEN
			Sollrichtung := 1;
		ELSE
			Sollrichtung := 0;
		END_IF
	END_IF	
ELSE
	Sollrichtung := 0;
END_IF
END_ACTION

END_FUNCTION_BLOCK

// ---- SRT_Allgemein/0010_Bausteine_mitDuts/POUs/FB_Automatik.TcPOU
FUNCTION_BLOCK FB_Automatik
VAR_INPUT
	in_frg_Safety	:BOOL;
	in_IBN		:BOOL;
END_VAR
VAR_OUTPUT
	out_Aktor_aktiv	:BOOL;
	out_frg_Automatik:BOOL;
END_VAR

VAR_IN_OUT
	inout_Steuerstatus	:DUT_Visu_SteuerStatus;
	sk								:INT;
END_VAR

VAR
END_VAR

//Automatik starten

IF inout_Steuerstatus.auto_start
THEN
	IF in_frg_Safety
	THEN
		inout_Steuerstatus.auto_aktiv:=TRUE;
	END_IF
	inout_Steuerstatus.auto_start:=FALSE;	
END_IF

//Automatik stoppen

IF inout_Steuerstatus.auto_stop
	OR inout_Steuerstatus.hand
THEN
		inout_Steuerstatus.auto_aktiv:=FALSE;
		inout_Steuerstatus.auto_stop:=FALSE;
END_IF

//Reset
	inout_Steuerstatus.grundstellung := inout_Steuerstatus.reset;
	
	IF inout_Steuerstatus.reset
	THEN
		out_Aktor_aktiv :=FALSE;
		GVL_1200.sk:=0;
		inout_Steuerstatus.grundstellung:=FALSE;
		inout_Steuerstatus.reset:=FALSE;
	END_IF
	
	//Freigabe Automatik
	out_frg_Automatik:=inout_Steuerstatus.auto_aktiv 
									AND (in_frg_Safety OR in_IBN);

END_FUNCTION_BLOCK

// ---- SRT_Allgemein/0010_Bausteine_mitDuts/POUs/FB_Bereichsueberwachung.TcPOU
FUNCTION_BLOCK FB_Bereichsueberwachung
VAR_INPUT
	/// Sollwert 
	in_sollwert: REAL;
	/// Istwert 
	in_istwert: REAL;
	/// Offset Obergrenze 
	in_offset_oben: REAL;
	/// Offset Untergrenze 
	in_offset_unten: REAL;
	/// Freigabe zum Überwachen 
	in_freigabe: BOOL;
END_VAR
VAR_OUTPUT
	/// Sollwerrt im Bereichsfenster (Sollwert= Istwert +/- Offset) 
	out_im_bereich: BOOL;
END_VAR
VAR
	temp_oben_real: REAL;
	temp_unten_real: REAL;
	temp_grenze_oben: BOOL;
	temp_grenze_unten: BOOL;
END_VAR

	(* Obergrenze überschritten ? *)
	temp_oben_real := in_sollwert +in_offset_oben;
	temp_grenze_oben := in_istwert > temp_oben_real;

	(* Untergrenze unterschritten ? *)
	temp_unten_real := in_sollwert - in_offset_unten;
	temp_grenze_unten := in_istwert < temp_unten_real;

	(* Wert liegt im zulässigen Bereich *)
	out_im_bereich := in_freigabe
					AND NOT temp_grenze_unten
					AND NOT temp_grenze_oben;

END_FUNCTION_BLOCK

// ---- SRT_Allgemein/0010_Bausteine_mitDuts/POUs/FB_FU_Rexroth.TcPOU
FUNCTION_BLOCK FB_FU_Rexroth
VAR_INPUT
	in_PD					:DUT_Rexroth_FU_PD_IN;
	in_NotHalt				:BOOL;	// 1=NotHalt aktiv
	in_Reset				:BOOL;	
	in_Auto_vor				:BOOL;	
	in_Auto_zur				:BOOL;	
	in_Auto_Drehzahl		:UINT;	
	in_Nenndrehzahl			:UINT;	
	in_Hand					:BOOL;	
END_VAR
VAR_OUTPUT
	out_PD					:DUT_Rexroth_FU_PD_OUT;
	out_Stoerung			:BOOL;	(* Umrichter meldet Störung *)
	out_Nicht_Bereit		:BOOL;	(* Umrichter ist nicht betriebsbereit *)
	out_Drehzahl_Ist		:INT;	(* aktuelle Drehzahl *)
	out_ist_90				:BOOL;	(* 90% der Soll Drehzahl erreicht *)
	out_Fehlernummer		:BYTE;	(* Fehlernummer *)
	out_Dreht				:BOOL;
END_VAR

VAR_IN_OUT
	inout_Visu_steuern			:DUT_SEW_FU_Visu;	(* Visu Steuerstruktur + *)
END_VAR

VAR
	VERZ_90_OK			:ton;
END_VAR

VAR_TEMP
	RECHTSLAUF				:BOOL;
	LINKSLAUF				:BOOL;
	TEMP_V					:REAL;
	TEMP_DREHZAHL_SOLL		:REAL;
END_VAR


(* Steuerwort --------------------------------------------------------------------*)
(*
Bit		Wert	Bedeutung
15…8 	-		Fehlercode
	--------------------------------------------------------------------------------
7		1		Fehler
		0		kein Fehler
	--------------------------------------------------------------------------------
6		1		Begrenzung Überstrom
		0		Normal
	--------------------------------------------------------------------------------
5		1		Begrenzung Überspannung
		0		Normal
	--------------------------------------------------------------------------------
4		1		Verzögerung
		0		keine Verzögerung
	--------------------------------------------------------------------------------
3		1		Beschleunigung
		0		keine Beschleunigung
	--------------------------------------------------------------------------------
2		1		Tippbetrieb
		0		kein Tippbetrieb
	--------------------------------------------------------------------------------
1		1		Start
		0		Stop
	--------------------------------------------------------------------------------
0		1		Rückwärts
		0		Vorwärts
*)

 //Störung *************************************************************************
	//out_Fehlernummer :=in_PD.PD_1_STATUSWORT.B1;

	IF NOT in_PD.PD_1_STATUSWORT.7 
	THEN
		out_Fehlernummer :=0;
	END_IF

	out_Stoerung	:=in_PD.PD_1_STATUSWORT.7 ;
// Bereit ***************************************************************************
	out_Nicht_Bereit:=in_PD.PD_1_STATUSWORT.7
						OR in_PD.PD_1_STATUSWORT.6
						OR in_PD.PD_1_STATUSWORT.5;
//Ausgabe ISt-Drehzahl***************************************************************
	out_Drehzahl_Ist				 :=WORD_TO_INT(in_PD.PD_2_IST_DREHZAHL)*(in_Nenndrehzahl/1000);
	
	inout_Visu_steuern.istdrehzahl	:=WORD_TO_INT(in_PD.PD_2_IST_DREHZAHL)*(in_Nenndrehzahl/1000);

	out_Dreht:=out_Drehzahl_Ist>10;

//	VERZ_90_OK(in:=out_Dreht AND out_PD.PD_1_Steuerwort.0,
//						pt:=T#9S);	
//	out_ist_90:=VERZ_90_OK.Q;	//ABS(out_Drehzahl_Ist) >ABS((temp_drehzahl_soll/100*90))
	out_ist_90:=ABS(out_Drehzahl_Ist) >ABS((temp_drehzahl_soll/100*90));

	
//Rechtslauf Hand-Automatik (mit Drehrichtungstausch)******************************************
	rechtslauf := ((inout_Visu_steuern.plus_start 
						AND in_HAnd)
				  OR(in_auto_vor 
						AND NOT IN_HAND ));
		
//Linkslauf Hand-Automatik (mit Drehrichtungstausch)****************************************
	linkslauf:=((inout_Visu_steuern.minus_stop 
						AND IN_HAND)
				  OR(in_auto_zur 
						AND NOT IN_HAND ));
	
//Geschwindigkeit umkopieren************************************************************
	IF IN_HAND 
	THEN 
		temp_v := inout_Visu_steuern.override/(in_Nenndrehzahl/1000);
		ELSE 
			temp_v := in_Auto_Drehzahl/(in_Nenndrehzahl/1000);
	END_IF
	
//Drehzahl ermitteln*************************************************************************
	temp_drehzahl_soll:= temp_v;

	IF temp_drehzahl_soll >= in_Nenndrehzahl
		THEN temp_drehzahl_soll:=in_Nenndrehzahl;
	END_IF

// -------------------------------------------------------------------------------------------
	// ---------------------------------------------------------------------------------------
	// Prozessdaten schreiben
	
	//Vorgabe Soll-Drehzahl--------------------------------------------------------------------
	out_PD.PD_2_solldrehzahl :=TO_UINT(temp_drehzahl_soll);

	//	Startbefehl----------------------------------------------------------------------------
	out_PD.PD_1_Steuerwort.0 := NOT in_NotHalt
								AND (linkslauf OR rechtslauf); 
	//	Tippbetrieb	----------------------------------------------------------------------------							
	out_PD.PD_1_Steuerwort.1 := NOT in_NotHalt
								AND IN_HAND
								AND inout_Visu_steuern.betriebsart=1;
	//	Vorwärts(0)/Rückwerts(1)----------------------------------------------------------------
	out_PD.PD_1_Steuerwort.2 := ((linkslauf 
										AND NOT in_Hand)                                                     
									OR IN_HAND   
										AND inout_Visu_steuern.betriebsart<>1                      
										AND (inout_Visu_steuern.minus_stop)) ;                     
	//	Stopp gemäß Parameter-------------------------------------------------------------------
	out_PD.PD_1_Steuerwort.3 := NOT linkslauf                                                   
								AND NOT rechtslauf;                                             
	//	Not-Aus (Not-Aus Rampe)	----------------------------------------------------------------
	out_PD.PD_1_Steuerwort.4 := in_NotHalt;                                                  
	//	Reset                                                                                   
	out_PD.PD_1_Steuerwort.5 := IN_RESET;                                                       
	//	Stop Beschl./Verz. mit internen Rampen--------------------------------------------------
	out_PD.PD_1_Steuerwort.6 := FALSE;                                                          
	//	Steuerwort aktivieren-------------------------------------------------------------------
	out_PD.PD_1_Steuerwort.7 := TRUE;                                                           
	//	Austrudeln------------------------------------------------------------------------------
	out_PD.PD_1_Steuerwort.8 := FALSE;                                                          
	//	Reserve---------------------------------------------------------------------------------
	out_PD.PD_1_Steuerwort.9  := FALSE;
	out_PD.PD_1_Steuerwort.10 := FALSE;
	out_PD.PD_1_Steuerwort.11 := FALSE;
	out_PD.PD_1_Steuerwort.12 := FALSE;
	out_PD.PD_1_Steuerwort.13 := FALSE;
	out_PD.PD_1_Steuerwort.14 := FALSE;
	out_PD.PD_1_Steuerwort.15 := FALSE;
	
(* Steuerwort --------------------------------------------------------------------*)
(*
Bit		Wert	Bedeutung
15…9 	-		Reserviert
	--------------------------------------------------------------------------------
8		1		Austrudeln
		0		Inaktiv
	--------------------------------------------------------------------------------
7		1		Steuerwort aktiv
		0		Inaktiv
	--------------------------------------------------------------------------------
6		1		Stopp Beschl./Verz. aktiv (stoppt den internen Beschleunigungs-/Verzögerungsrampengenerator)
		0		Inaktiv
	--------------------------------------------------------------------------------
5		1		Fehler Rücksetzen aktiv
		0		Inaktiv
	--------------------------------------------------------------------------------
4		1		Not-Aus aktiv
		0		Inaktiv
	--------------------------------------------------------------------------------
3		1		Stopp gemäß Parametereinstellung
		0		Inaktiv
	--------------------------------------------------------------------------------
2		1		Rückwärts
		0		Vorwärts
	--------------------------------------------------------------------------------
1		1		Tippbetrieb aktiv (Schrittrichtung bestimmt durch Bit 2)
		0		Inaktiv
	--------------------------------------------------------------------------------
0		1		Startbefehl aktiv
		0		Inaktiv

*)

END_FUNCTION_BLOCK

// ---- SRT_Allgemein/0010_Bausteine_mitDuts/POUs/FB_Messachse_EL3051.TcPOU
FUNCTION_BLOCK FB_Messachse_EL3051
VAR_INPUT
	in_EncPos				: INT;
	in_min_sensor			: INT;	(*minimal Wert vom Sensor*)
	in_max_sensor			: INT;	(*maximal Wert vom Sensor*)
	in_min_norm				: REAL;	(*minimal zu normierenden Wert z.B. 0% oder 25mm *)
	in_max_norm				: REAL;	(*maximal zu normierenden Wert z.B. 100% oder 1025mm*)
	in_OffsetIstPos			: LREAL;
    in_bPneumatikCommand 	: BOOL;           // TRUE wenn Vorschubbefehl aktiv
END_VAR
VAR_OUTPUT
	out_IstPos				: LREAL;
	out_bDone				: BOOL;	// Ref Position ist gesetzt worden
	out_bValid				: BOOL; // Positionwert ist stabil
END_VAR
VAR
	temp_Pos				: LREAL;
	RT_SetPos				: R_TRIG;
	ton_Valid				: ton;
	
	EncoderPos      : LINT;     // akt. Encoderposition (lesen)
    EncoderPosPrev  : LINT := 0;
    Delta           : LINT;
    DeadbandCounts  : LINT := 9;        // hier: ~0.1 mm -> 9 counts
    SampleTimeMs    : TIME := T#10MS;   // Zykluszeit (zur Info)
    StableTimer     : TON;
    StableTimePT    : TIME := T#200MS;  // Bestätigungszeit
    bStableCount    : BOOL;
    bAnschlagGefunden : BOOL;           // Ausgang: Anschlag erkannt
	temp_min_sensor		:REAL;
	temp_max_sensor		:REAL;
	temp_out			:REAL;
	temp_in_sensor		:REAL;
	temp_diff			:REAL;
END_VAR

// Istposition umrechnen in eine Einheit

	(* Eingänge wandeln *)
	temp_min_sensor	:=INT_TO_REAL(in_min_sensor);
	temp_max_sensor	:=INT_TO_REAL(in_max_sensor);
	temp_in_sensor	:=INT_TO_REAL(in_EncPos);
	
	(* Messwerte normieren und ausgeben *)
	temp_out:=	(((in_max_norm-in_min_norm) 					(* Normbereich ermitteln *)
						/ (temp_max_sensor - temp_min_sensor))	(* Messbereich ermitteln *)
				* (temp_in_sensor-temp_min_sensor));			(* Eingange des Messsensors *)
	(*  *)						
	 out_IstPos :=(in_min_norm + temp_out + in_OffsetIstPos);

// Stabile Position erkannt
// --- Hauptlogik (zyklisch) ---
	EncoderPos := in_EncPos; // 
	
	Delta := ABS(EncoderPos - EncoderPosPrev);
	
	IF Delta <= DeadbandCounts THEN
		bStableCount := TRUE;
	ELSE
		bStableCount := FALSE;
	END_IF
	
	// TON nutzt die Eingangssignallogik
	StableTimer(IN := bStableCount, PT := StableTimePT);
	
	// Anschlag nur, wenn Position stabil *und* Pneumatikbefehl noch aktiv (optional)
	IF StableTimer.Q AND in_bPneumatikCommand THEN
		out_bValid := TRUE;
	ELSE
		out_bValid := FALSE;
	END_IF
	
	EncoderPosPrev := EncoderPos;

END_FUNCTION_BLOCK

// ---- SRT_Allgemein/0010_Bausteine_mitDuts/POUs/FB_Schutztuer_mitBremsentest.TcPOU
FUNCTION_BLOCK FB_Schutztuer_mitBremsentest
(*
	Ansteuerung der Schutztüren mit anstoßen des Bremsentests 
	Autor O.E.
	Erstellt 06.09.2022
	Version 1.0 	
*)
VAR_INPUT
	in_Anfordern_Quitt		:BOOL;(*Anforderungstaster Schutztür öffnen / Ablauf Reset=5Sek gedrückt*)             
	in_Ablauf_Start			:BOOL;(*Ablauf wieder starten*) 
	in_Steuerhilfsluft		:BOOL;            
	in_Tuer_zu				:BOOL;(*Schutztür geschlossen            *)               
	in_Tuer_verriegelt		:BOOL;(*Schutztür geschlossen und verriegelt*)                           
	in_frg_zutritt			:BOOL;(*Anlagenzyklus steht, Freigabe Zutritt*)    
	in_2mal_anfordern		:BOOL;(*es muss innerhalb von 3Sekunden zweimal die Anfordern-Taste gedrückt werden*)
	in_mit_bremsentest		:BOOL;(*mit Bremsentest?  0=nein, 1=ja*)
    in_bremsentest_ok		:BOOL;(*Bremsentest ok/fehlerfrei*)
 
END_VAR
VAR_OUTPUT
	out_Tuer_entr_high		:BOOL;(*Schutztür entriegeln im Ruhezustand 1*)
	out_Tuer_entr_low		:BOOL;(*Schutztür entriegeln im Ruhezustand 0*)
	out_Led_Anf_quitt		:BOOL;(*Meldeleuchte Schutztür*)
	out_Led_Ablauf_start	:BOOL;(*Meldeleuchte Schutztür*)
	out_Freigabe			:BOOL;(*Türen Freigeben*)
	out_Zyk_stop			:BOOL;(*Zyklus anhalten*)
END_VAR

VAR_IN_OUT
	inout_bremsentest_start	:BOOL;(*Bremsentest starten*)	
END_VAR

VAR
	sk						:INT;(*Schrittkette*)
	totzeit					:TON;(*Totzeit nach erster Anforderung*)
	verz_reset				:ton;
	fl_bremsentest			:r_trig;(**)
	fl_Anfordern			:R_TRIG;
	nFl_Anfordern			:F_TRIG;			
	t_100ms_an				:ton;
	t_100ms_aus				:tof;
	
	t_500ms_an				:ton;
	t_500ms_aus				:tof;
	
	t_1000ms_an				:ton;
	t_1000ms_aus			:tof;
	
END_VAR

//***** Sondersachen, Zeiten Berechnungen oder was auch immer **************************************************
	//**********************************************************************************************************
	
	
totzeit(PT:=  T#60S,
		IN:=(sk=30 AND NOT inout_bremsentest_start)
				OR(sk=40 AND in_Tuer_zu));
verz_reset(pt:=T#5S,
			in:= in_Anfordern_Quitt);
			
fl_Anfordern(clk:=in_Anfordern_Quitt);		
nFl_Anfordern(CLK:=in_Anfordern_Quitt);

t_100ms_an(IN:=NOT t_100ms_aus.Q , PT:=T#100MS);
t_100ms_aus(IN:=t_100ms_an.Q , PT:=T#100MS , Q=>);
	
t_500ms_an(IN:=NOT t_500ms_aus.Q , PT:=T#500MS);
t_500ms_aus(IN:=t_500ms_an.Q , PT:=T#500MS , Q=>);
	
t_1000ms_an(IN:=NOT t_1000ms_aus.Q , PT:=T#1000MS);
t_1000ms_aus(IN:=t_1000ms_an.Q , PT:=T#1000MS , Q=>);
	
//***** Reset **************************************************************************************************
	//**********************************************************************************************************
IF verz_reset.Q
	OR totzeit.Q
THEN
	sk							:= 0;
END_IF

//***** P r o g r a m m   S t a r t ****************************************************************************
	//**********************************************************************************************************
CASE sk OF

	0:// Schritt 0 fangen wir an Start Schrittkette 
		IF fl_Anfordern.Q
		THEN
			sk		:= 10;
		END_IF
		
		IF NOT in_Anfordern_Quitt
			AND (NOT in_Tuer_zu
				OR NOT in_Tuer_verriegelt)
		THEN
			sk		:= 50;
		END_IF
		
	10:// Schritt 10 Anforderungstaster gelöst 
		IF NOT in_Anfordern_Quitt
			AND NOT in_2mal_anfordern
		THEN
			sk		:= 30;
		END_IF

		IF NOT in_Anfordern_Quitt
			AND in_2mal_anfordern
		THEN
			sk		:= 20;
		END_IF

	20:// Schritt 20 Zweite Betätigung Anforderungstaster  
		IF in_Anfordern_Quitt
		THEN
			sk		:= 30;
		END_IF
		
	30:// Schritt 30 Schutztür entriegeln  
		IF NOT in_Anfordern_Quitt
			AND in_frg_zutritt
			AND (NOT in_mit_bremsentest
				OR in_bremsentest_ok)
		THEN
			sk		:= 40;
		END_IF

	40:// Schritt 40 Schutztür ist offen  
		IF NOT in_Tuer_zu
			OR in_Tuer_verriegelt
		THEN
			sk		:= 50;
		END_IF

	50:// Schritt 50 Anforderung Schutztür verriegeln 
		IF in_Tuer_zu
			AND NOT in_Tuer_verriegelt
			AND in_Anfordern_Quitt
		THEN
			sk		:= 60;
		END_IF

	60:// Schritt 60 Schutztür ist verriegelt 
		IF in_Tuer_zu
			AND in_Tuer_verriegelt
			AND NOT in_Anfordern_Quitt
		THEN
			sk		:= 70;
		END_IF

	70:// Schritt 70 Ablauf start
		IF in_Tuer_zu
			AND in_Tuer_verriegelt
			AND in_Ablauf_Start
		THEN
			sk		:= 80;
		END_IF
		
		IF nFl_Anfordern.Q
			AND in_Tuer_verriegelt
			AND in_Tuer_zu
		THEN
			sk		:= 10;
		END_IF
		
	80:// Schritt 80 
		IF in_Tuer_zu
			AND in_Tuer_verriegelt
			AND NOT in_Ablauf_Start
		THEN
			sk		:= 0;
		END_IF

END_CASE

//***** Ausgaenge **********************************************************************************************
	//**********************************************************************************************************
	
	//***** Meldeleuchte Anforderung ***************************************************************************
		//******************************************************************************************************
	out_Led_anf_quitt 	:= ((sk = 10  
								OR sk = 20 
								OR (sk = 30 AND t_1000ms_aus.q)
								OR (sk = 40 AND t_500ms_aus.q)
								OR (sk = 50 AND t_500ms_aus.Q)
								OR sk = 60 
								OR sk = 70  
								OR sk = 80 )
								AND NOT in_Steuerhilfsluft)
							OR (in_Steuerhilfsluft
										AND NOT out_Led_Ablauf_start)
							OR (sk = 0  AND in_Tuer_verriegelt AND in_Tuer_zu);
							
	out_Led_Ablauf_start:=	(((sk = 70 AND t_500ms_aus.Q)  
								OR 	sk = 80)
								AND NOT in_Steuerhilfsluft)
							OR  (in_Steuerhilfsluft
								AND t_100ms_aus.q
								AND	(NOT in_Tuer_verriegelt));
													
		
	//***** Schutztür entriegeln *******************************************************************************
		//******************************************************************************************************
	out_Tuer_entr_low :=NOT	( sk = 40 
							OR sk = 50);
	out_Tuer_entr_high :=	( sk = 40 
							OR sk = 50);
	
	//***** Bremsentest start  *********************************************************************************
		//******************************************************************************************************
	fl_bremsentest(clk:=in_mit_bremsentest
						AND in_frg_zutritt
						AND sk = 30);
	IF fl_bremsentest.Q
	THEN
		inout_bremsentest_start:=TRUE;
	END_IF
		
	//***** Zyklus anhalten ************************************************************************************
		//******************************************************************************************************
	out_Zyk_stop:= sk>20
					AND sk<80;
					
	out_Freigabe:=	sk>30
					AND sk<80;
//EndeEndeEndeEndeEndeEndeEndeEndeEndeEndeEndeEndeEndeEndeEndeEndeEndeEndeEndeEndeEndeEndeEndeEndeEndeEndeEndeE*)

END_FUNCTION_BLOCK

// ---- SRT_Allgemein/0010_Bausteine_mitDuts/POUs/FB_Ventil.TcPOU
FUNCTION_BLOCK FB_Ventil
(*
	Ansteuerungsbaustein zum Steuern und Überwachen von Ventilen und den dazugehörigen Sensoren
	(abgeleitet vom Siemens Baustein "Allg-Ventilbaustein" Stand 20.01.20)
	Autor O.E.
	Erstellt 20.01.20
	Version 1.0 
*)
VAR_INPUT
	in_endlage_vor	:BOOL;	(*1=Endlage vorne ist angefahren*)
	in_endlage_zur	:BOOL;	(*1=Endlage zurück ist angefahren*)
	in_hand			:BOOL;	(*1=Handbetrieb*)
	in_auto			:BOOL;	(*1=Automatikbetrieb*)
	in_quit			:BOOL;	(*		*)
END_VAR

VAR_OUTPUT
	out_vor				:BOOL;				(*Ausgang vorfahren*)
	out_zur				:BOOL;				(*Ausgang zurückfahren*)
	out_stoerung_vor	:BOOL;				(*Störung*)
	out_stoerung_zur	:BOOL;				(*Störung*)
	out_stoerung_vorzur	:BOOL;				(*Störung*)
	out_vor_visu		:BOOL;				(*Endlagen direkt für die Visu weitergeleitet*)
	out_zur_visu		:BOOL;				(*Endlagen direkt für die Visu weitergeleitet*)
END_VAR

VAR_IN_OUT
	inout_ansteuerung	:DUT_Ventil_sps;
	inout_visu			:DUT_Ventil_VISU;
END_VAR

VAR
	temp_zeit_vor				:TIME;
	temp_zeit_zur				:TIME;
	temp_zeit_entprellen_vor	:TIME;
	temp_zeit_entprellen_zur	:TIME;
	temp_end_vor				:BOOL;
	temp_end_zur				:BOOL;
	temp_stoer_vor				:BOOL;
	temp_stoer_zur				:BOOL;
	temp_stoer_vor_zur			:BOOL;	
END_VAR

VAR	
	verzoegerung_vor			:TON;	
	verzoegerung_zur			:TON;		
	ueberwachung_vor			:TON;		
	ueberwachung_zur			:TON;	
	fl_hm_vor					:R_trig;	
	fl_hm_zur					:R_trig;	

	hm_vor						:BOOL;	
	hm_zur						:BOOL;	
	hm_timer_reset				:BOOL;	
	hm_timer_reset_2			:BOOL;	
END_VAR

(************************************************************************************************************************************************************)
(*	SIGNALE IN 
		in_endlage_vor		--- 1 = Endlage vorne ist angefahren
		in_endlage_zur		--- 1 = Endlage zurück ist angefahren
		in_hand				--- Handbetrieb
		in_auto				--- Automatikbetrieb
		in_quit				--- Störungs Reset
						
	SIGNALE OUT 
		out_vor				--- Ausgang vorfahren
		out_zur				--- Ausgang zurückfahren
		out_stoerung		--- Störung
	
	SIGNALE INOUT - SPS
		in_auto_vor			--- Startsignal vorfahren (bleibt gespeichert)
		in_auto_zur			--- Startsignal zurückfahren (bleibt gespeichert)
		in_aus				--- intern gespeicherte Startsignale löschen
		in_freigabe_vor		--- 1 = vorfahren freigegeben
		in_freigabe_zur		--- 1 = zurückfahren freigegeben
		
		out_ist_vor			--- steht in Endlage vor und kein Fehler
		out_ist_zur			---	steht in Endlage zur und kein Fehler
	
	SIGNALE INOUT - VISU
		hand_vor			--- Hand vorfahren
		hand_zur			--- Hand zurückfahren
		reset				--- ntern gespeicherte Startsignale löschen
		service				--- 1 = ALLE Überwachungen deaktiviert
		status				--- 0=??? 1=vor 2=ist vor 3=fehler vor 4=zur 5=ist zur 6=Fehler zur 7=Fehler vor zur
		para				--- Parameter Struktur
			ueberwachung_vor_aktiv	--- 0 = Endlagenüberwachung vor deaktiviert
			ueberwachung_zur_aktiv	--- 0 = Endlagenüberwachung zurück deaktiviert
			ausgang_vor_halten		--- 1 = Ausgang immer Ein, sonst 0 in Endlage/1 nicht in Endlage
			ausgang_zur_halten		--- 1 = Ausgang immer Ein, sonst 0 in Endlage/1 nicht in Endlage
			entprellen_vor_aktiv	--- 0 = Endlage sofort überwachen wenn einmal erreicht
			entprellen_zur_aktiv	--  0 = Endlage sofort überwachen wenn einmal erreicht
			ueberwachungszeit_vor	--- Überwachungszeit in ms (0-30000ms)
			ueberwachungszeit_zur	--- Überwachungszeit in ms (0-30000ms)
			entprellungszeit_vor	--- Entprellungszeit in ms (0-10000ms)
			entprellungszeit_zur	--- Entprellungszeit in ms (0-10000ms)																					*)
(************************************************************************************************************************************************************)


(****** Zeitvorgabe prüfen **********************************************************************************************************************************)
(* Überwachung vor -> 0-300000ms  *)
	temp_zeit_vor:=inout_visu.para.ueberwachungszeit_vor;
	IF temp_zeit_vor<T#0MS
	THEN
		temp_zeit_vor:=T#0MS;
	END_IF
	
	IF temp_zeit_vor>T#30000MS
	THEN
		temp_zeit_vor:=T#30000MS;
	END_IF
(* Überwachung zurück -> 0-300000ms *)
	temp_zeit_zur:=inout_visu.para.ueberwachungszeit_zur;
	IF temp_zeit_zur<T#0MS
	THEN
		temp_zeit_zur:=T#0MS;
	END_IF
	
	IF temp_zeit_zur>T#30000MS
	THEN
		temp_zeit_zur:=T#30000MS;
	END_IF
(* Entprellen vor -> 0-10000s *)
	temp_zeit_entprellen_vor:=inout_visu.para.entprellungszeit_vor;
	IF temp_zeit_entprellen_vor<T#0MS
	THEN
		temp_zeit_entprellen_vor:=T#0MS;
	END_IF
	
	IF temp_zeit_entprellen_vor>T#10000MS
	THEN
		temp_zeit_entprellen_vor:=T#10000MS;
	END_IF
(* Entprellen zurück -> 0-10000ms *)
	temp_zeit_entprellen_zur:=inout_visu.para.entprellungszeit_zur;
	IF temp_zeit_entprellen_zur<T#0MS
	THEN
		temp_zeit_entprellen_zur:=T#0MS;
	END_IF
	
	IF temp_zeit_entprellen_zur>T#10000MS
	THEN
		temp_zeit_entprellen_zur:=T#10000MS;
	END_IF
(****** Endlage vor **********************************************************************************************************************************)
	verzoegerung_vor(IN:= in_endlage_vor
						AND NOT in_endlage_zur
						AND NOT hm_zur
						AND hm_timer_reset,
						pt:= temp_zeit_entprellen_vor);
	temp_end_vor:=((verzoegerung_vor.Q
					AND NOT inout_visu.service)
					OR (hm_vor
						AND inout_visu.service));
(****** Endlage zur **********************************************************************************************************************************)
	verzoegerung_zur(IN:= in_endlage_zur
						AND NOT in_endlage_vor
						AND NOT hm_vor
						AND hm_timer_reset,
						pt:= temp_zeit_entprellen_zur);
	temp_end_zur:=((verzoegerung_zur.Q
					AND NOT inout_visu.service)
					OR (hm_zur
						AND inout_visu.service));
(****** Start vor **********************************************************************************************************************************)
	IF ((in_auto
			AND inout_ansteuerung.in_auto_vor)
		OR (in_hand
			AND inout_visu.hand_vor))
		AND inout_ansteuerung.in_freigabe_vor
		AND NOT inout_ansteuerung.in_aus
	THEN
		hm_vor:=TRUE;
	END_IF
	
	IF (in_auto
			AND inout_ansteuerung.in_auto_zur)
		OR (in_hand
			AND inout_visu.hand_zur)
		OR inout_visu.reset
		OR inout_ansteuerung.in_aus
	THEN
		hm_vor:=FALSE;
	END_IF
	
	out_vor:=hm_vor
				AND inout_ansteuerung.in_freigabe_vor
				AND (NOT temp_end_vor
						OR inout_visu.para.ausgang_vor_halten);

(****** Start zur **********************************************************************************************************************************)
	IF ((in_auto
			AND inout_ansteuerung.in_auto_zur)
		OR (in_hand
			AND inout_visu.hand_zur))
		AND inout_ansteuerung.in_freigabe_zur
		AND NOT inout_ansteuerung.in_aus
	THEN
		hm_zur:=TRUE;
	END_IF

	IF (in_auto
			AND inout_ansteuerung.in_auto_vor)
		OR (in_hand
			AND inout_visu.hand_vor)
		OR inout_visu.reset
		OR inout_ansteuerung.in_aus
	THEN
		hm_zur:=FALSE;
	END_IF
	
	out_zur:=hm_zur
				AND inout_ansteuerung.in_freigabe_zur
				AND (NOT temp_end_zur
						OR inout_visu.para.ausgang_zur_halten);

(****** Flankenbildung bei vor und zurück *************************************************************************************************************)
(*wird benötigt damit der Timer bei direkten umschalten neu startet*) 
	fl_hm_vor(CLK:=hm_vor);
	fl_hm_zur(CLK:=hm_zur);
	
	hm_timer_reset_2:=fl_hm_vor.Q
					OR fl_hm_zur.Q
					OR ( NOT hm_vor
							AND NOT hm_zur)
					OR NOT inout_visu.para.ueberwachung_vor_aktiv	
					OR NOT inout_visu.para.ueberwachung_zur_aktiv	
					OR (out_stoerung_vorzur
						AND (temp_end_vor
								OR temp_end_zur))
					OR (hm_vor
						AND temp_end_vor)			
					OR (hm_zur
						AND temp_end_zur);			
	
(****** Zeitüberwachung Vor starten  *************************************************************************************************************)
	ueberwachung_vor(IN:=inout_visu.para.ueberwachung_vor_aktiv
							AND hm_vor
							AND NOT hm_timer_reset_2,
						pt:=temp_zeit_vor);
		
(****** Zeitüberwachung Zur starten  *************************************************************************************************************)
	ueberwachung_zur(IN:=inout_visu.para.ueberwachung_zur_aktiv
							AND hm_zur
							AND NOT hm_timer_reset_2,
						pt:=temp_zeit_zur);
		
(****** Störung - Zeitüberwachung Vor abgelaufen = Fehler *****************************************************************************************)
	temp_stoer_vor:=ueberwachung_vor.Q
					AND NOT temp_end_vor;
				
(****** Störung - Zeitüberwachung Zurück abgelaufen = Fehler **************************************************************************************)
	temp_stoer_zur:=ueberwachung_zur.Q
					AND NOT temp_end_zur;
	
(****** Störung - Beide Endlagen belegt = Fehler ***************************************************************************************************)
	temp_stoer_vor_zur:=temp_stoer_vor
						AND temp_stoer_zur;

(****** Störung - Ausgabe - STATUS auf 0 ************************************************************************************************************)
	IF in_quit
	THEN
		hm_timer_reset_2		:=FALSE;
		inout_visu.status		:=0;
	 	out_stoerung_vorzur		:=FALSE;
		out_Stoerung_vor		:=FALSE;
		out_Stoerung_zur		:=FALSE;
	END_IF						

	IF temp_stoer_vor
		AND NOT temp_stoer_vor_zur
	THEN
	 	out_stoerung_vor:=TRUE;
	END_IF						

	IF temp_stoer_zur
		AND NOT temp_stoer_vor_zur
	THEN
	 	out_stoerung_zur:=TRUE;
	END_IF						

	IF temp_stoer_vor_zur
	THEN
	 	out_stoerung_vorzur:=TRUE;
	END_IF						

	
(****** steht in Endlage vor und kein Fehler ********************************************************************************************************)
	inout_ansteuerung.out_ist_vor:= NOT out_stoerung_vorzur
									AND temp_end_vor;

(****** steht in Endlage zurück und kein Fehler *****************************************************************************************************)
	inout_ansteuerung.out_ist_zur:= NOT out_stoerung_vorzur
									AND temp_end_zur;
									
(***** Status ****************************************************************************************************************************************)
	(* 1=vor *)							
	IF hm_vor
		AND NOT temp_end_vor
		AND NOT temp_stoer_zur
		AND NOT temp_stoer_vor_zur
	THEN
		inout_visu.status:=1;									
	END_IF									
	(* 2=ist vor *)							
	IF (temp_end_vor
		OR (NOT inout_visu.para.ueberwachung_vor_aktiv
				AND hm_vor))
		AND NOT temp_end_zur
		AND NOT temp_stoer_zur
		AND NOT temp_stoer_vor_zur
	THEN
		inout_visu.status:=2;									
	END_IF															
	(* 3=Fehler vor	*)							
	IF temp_stoer_vor
	THEN
		inout_visu.status:=3;
	END_IF
	
	(* 4=zur *)							
	IF hm_zur
		AND NOT temp_end_zur
		AND NOT temp_stoer_zur
		AND NOT temp_stoer_vor_zur
	THEN
		inout_visu.status:=4;									
	END_IF									
	(* 5=ist zur *)							
	IF (temp_end_zur
		OR (NOT inout_visu.para.ueberwachung_zur_aktiv
				AND hm_zur))
		AND NOT temp_end_vor
		AND NOT temp_stoer_zur
		AND NOT temp_stoer_vor_zur
	THEN
		inout_visu.status:=5;									
	END_IF															
	(* 6=Fehler zurück *)								
	IF temp_stoer_zur
	THEN
		inout_visu.status:=6;
	END_IF
	(* 7=Fehler vor zur	*)
	IF temp_stoer_vor_zur
	THEN
		inout_visu.status:=7;
	END_IF

	
(***** Endlagen direkt an die Visu weiter reichen ***********************************************************************************************************)
	out_vor_visu:=in_endlage_vor;
	out_zur_visu:=in_endlage_zur;


(***** IN Start-Befehle Hand und Automatik löschen **********************************************************************************************************)
	inout_ansteuerung.in_auto_vor:=FALSE;
	inout_ansteuerung.in_auto_zur:=FALSE;
	inout_ansteuerung.in_aus := FALSE;
	inout_visu.hand_vor:=FALSE;
	inout_visu.hand_zur:=FALSE;
	hm_timer_reset:=TRUE;

END_FUNCTION_BLOCK

// ---- SRT_Allgemein/0010_Bausteine_mitDuts/POUs/FC_Bereichsueberwachung.TcPOU
FUNCTION FC_Bereichsueberwachung : BOOL
VAR_INPUT
	/// Sollwert 
	in_sollwert: REAL;
	/// Istwert 
	in_istwert: REAL;
	/// Offset Obergrenze 
	in_offset_oben: REAL;
	/// Offset Untergrenze 
	in_offset_unten: REAL;
	/// Freigabe zum Überwachen 
	in_freigabe: BOOL;
END_VAR
VAR
	temp_oben_real: REAL;
	temp_unten_real: REAL;
	temp_grenze_oben: BOOL;
	temp_grenze_unten: BOOL;
END_VAR

	(* Obergrenze überschritten ? *)
	temp_oben_real := in_sollwert +in_offset_oben;
	temp_grenze_oben := in_istwert > temp_oben_real;

	(* Untergrenze unterschritten ? *)
	temp_unten_real := in_sollwert - in_offset_unten;
	temp_grenze_unten := in_istwert < temp_unten_real;

	(* Wert liegt im zulässigen Bereich *)
	FC_Bereichsueberwachung := in_freigabe
								AND NOT temp_grenze_unten
								AND NOT temp_grenze_oben;

END_FUNCTION

// ---- SRT_Allgemein/0010_Bausteine_mitDuts/POUs/FC_InRange.TcPOU
FUNCTION FC_InRange : BOOL
VAR_INPUT
	Soll: REAL;
	Ist: REAL;
	Range: REAL;
END_VAR
VAR
	temp_oben_real: REAL;
	temp_unten_real: REAL;
	temp_grenze_oben: BOOL;
	temp_grenze_unten: BOOL;
END_VAR

	(* Obergrenze überschritten ? *)
	temp_oben_real := Soll + (Range / 2);
	temp_grenze_oben := Ist > temp_oben_real;

	(* Untergrenze unterschritten ? *)
	temp_unten_real := Soll - (Range / 2);
	temp_grenze_unten := Ist < temp_unten_real;

	(* Wert liegt im zulässigen Bereich *)
	FC_InRange := 	NOT temp_grenze_unten
					AND NOT temp_grenze_oben;

END_FUNCTION

// ---- SRT_Allgemein/0010_Bausteine_mitDuts/POUs/FU_SEW/Movi_B/FB_SEW_MOVITRAC.TcPOU
FUNCTION_BLOCK FB_SEW_MOVITRAC
VAR_INPUT
	in_PD					:DUT_SEW_FU_PD_IN;
	in_Reglersperre			:BOOL;	(* 1= Regler sperren *)
	in_Dreh_Tausch			:BOOL;	(* Drehrichtung tauschen *)
	in_Rechts				:BOOL;	(* 1= Antrieb rechtslauf  (IN_hand=0) *)
	in_Links				:BOOL;	(* 1= Antrieb linkslauf (IN_hand=0) *)
	in_Reset				:BOOL;	(* 0->1 Fehler löschen *)
	in_Hand					:BOOL;	(* Hand aktiv *)
	in_Hand_rechts			:BOOL;	(* Softkey Motor Tippen + *)
	in_Hand_links			:BOOL;	(* Softkey Motor Tippen - *)
	in_Hand_V				:REAL;	(* Geschwindigkeit in m/min für Hand  *)
	in_V					:REAL;	(* Geschwindigkeit in m/min für Auto *)
	in_Rampe				:INT;	(* Rampe Hochlauf/Ablauf in ms *)
	V_Faktor				:REAL;	(* Drehzahlbezug (z.B. bei 1500 sec-1  /  30m/min  =  Faktor 50) *)
END_VAR
VAR_OUTPUT
	out_PD					:DUT_SEW_FU_PD_OUT;
	out_Stoerung			:BOOL;	(* Umrichter meldet Störung *)
	out_Nicht_Bereit		:BOOL;	(* Umrichter ist nicht betriebsbereit *)
	out_Drehzahl_Ist		:REAL;	(* aktuelle Drehzahl *)
	out_ist_90				:BOOL;	(* 90% der Soll Drehzahl erreicht *)
	out_Fehlernummer		:BYTE;	(* Fehlernummer *)
	out_Dreht				:BOOL;
	//OUT_WARNUNG				:BOOL;
END_VAR
VAR_TEMP
	reglersperre			:BOOL;	(* BIT 0: Reglersperre 0 = Freigabe 1 = Regler sperren, Bremse aktivieren *)
	freigabe_stop			:BOOL;	(* BIT 1: Freigabe/Schnellstopp 0 = Schnellstopp 1 = Freigabe *)
	freigabe_halt			:BOOL;	(* BIT 2: Freigabe/Halt 0 = Halt an Integratorrampe oder Prozess-Rampe 1 = Freigabe *)
	reserve_3_1				:BOOL;	(* BIT 3: Reserviert (Reservierte Bits sind generell auf Null zu setzen!) *)
	reserve_4_1				:BOOL;	(* BIT 4: Reserviert (Reservierte Bits sind generell auf Null zu setzen!) *)
	reserve_5_1				:BOOL;	(* BIT 5: Reserviert (Reservierte Bits sind generell auf Null zu setzen!) *)
	reset					:BOOL;	(* Bit 6: Reset 0 = nicht aktiv 0 -> 1 = anstehende Störung zurücksetzen *)
	reserve_7_1				:BOOL;	(* BIT 7: Reserviert (Reservierte Bits sind generell auf Null zu setzen!) *)
	drehrichtung_motorpoti	:BOOL;	(* BIT 8: Drehrichtung für Motorpoti 0 = Drehrichtung RECHTS 1 = Drehrichtung LINKS *)
	motorpoti_auf			:BOOL;	(* BIT 9 und 10: Motorpoti Hochlauf,Motorpoti Tieflauf 0 0 = keine Änderung *)
	motorpoti_ab			:BOOL;	(*  1 0 = ab 0 1 = auf 1 1 = keine Änderung *)
	n11_n21					:BOOL;	(* BIT 11 und 12:Anwahl der internen Festsollwerte0 0 = Drehzahl-Sollwert über Prozess-Ausgangsdatenwort 2 *)
	n12_n22					:BOOL;	(* 0 1 = interner Sollwert n11 (n21) *)
	sollwert_umschaltung	:BOOL;	(* BIT 13: Festsollwert-Umschaltung 0 = Festsollwerte des aktivn Parameter über Bit 11/12 anwählbar 1 = Festsollwerte des anderen Parameter anwählbar *)
	reserve_14				:BOOL;	(* BIT 14: Reserviert (Reservierte Bits sind generell auf Null zu setzen!) *)
	reserve_15				:BOOL;	(* BIT 14: Reserviert (Reservierte Bits sind generell auf Null zu setzen!) *)
	DREHZAHL				:REAL;
	RECHTSLAUF				:BOOL;
	LINKSLAUF				:BOOL;
	TEMP_V					:REAL;
	TEMP_IST_DREHZAHL_DINT	:DINT;
	TEMP_DREHZAHL			:REAL;
	TEMP_DREHZAHL_SOLL		:REAL;
	endstufe_freigeben		:BOOL;	(* BIT 0: Endstufe freigegeben 0 = Endstufe ist gesperrt (hochohmig) 1 = Endstufe ist freigegeben *)
	umrichter_bb			:BOOL;	(* BIT 1: Umrichter betriebsbereit 0 = Umrichter nicht betriebsbereit (z. B. Fehler) 1 = Umrichter betriebsbereit *)
	pa_daten_freigeben		:BOOL;	(* BIT 2: PA-Daten freigegeben 0 = PA-Daten gesperrt 1 = PA-Daten freigegeben *)
	reserve_3				:BOOL;	(*  Reserve Bit ist immer auf null zusetzen *)
	reserve_4				:BOOL;	(*  Reserve Bit ist immer auf null zusetzen *)
	stoerung				:BOOL;	(*  BIT 5: Störung/Warnung 0 = keine Störung/Warnung 1 = Störung/Warnung liegt an *)
	reserver_6				:BOOL;	(*  Reserve Bit ist immer auf null zusetzen *)
	fehlernummer			:BYTE;	(*  Byte 2: Gerätezustand/ Fehlernummer *)
	steuerbyte_1			:BYTE;
	steuerbyte_2			:BYTE;
END_VAR


//Statuswort auslesen*****************************************************************************************
	endstufe_freigeben 	:= BIT_OF_dWORD(in:= in_PD.PD_1_STATUSWORT, N:= 0);
	umrichter_bb 		:= BIT_OF_dWORD(in:= in_PD.PD_1_Statuswort, N:= 1);
	pa_daten_freigeben	:= BIT_OF_DWORD(in:= in_PD.PD_1_Statuswort, N:= 2);
	reserve_3			:= BIT_OF_DWORD(in:= in_PD.PD_1_Statuswort, N:= 3);
	reserve_4			:= BIT_OF_DWORD(in:= in_PD.PD_1_Statuswort, N:= 4);
	stoerung			:= BIT_OF_DWORD(in:= in_PD.PD_1_Statuswort, N:= 5);
	reserver_6 			:= BIT_OF_DWORD(in:= in_PD.PD_1_Statuswort, N:= 6);
	fehlernummer		:= BYTE_OF_DWORD(in:= in_PD.PD_1_Statuswort, N:= 1);
(*Statuswort  --------------------------------------------------------------------
	BIT 0: Endstufe freigegeben
	0 = Endstufe ist gesperrt (hochohmig)
	1 = Endstufe ist freigegeben
	--------------------------------------------------------------------------------
	BIT 1: Umrichter betriebsbereit
	0 = Umrichter nicht betriebsbereit (z. B. Fehler)
	1 = Umrichter betriebsbereit
	--------------------------------------------------------------------------------
	BIT 2: PA-Daten freigegeben
	0 = PA-Daten gesperrt
	1 = PA-Daten freigegeben
	--------------------------------------------------------------------------------
	BIT 5: Störung/Warnung
	0 = keine Störung/Warnung
	1 = Störung/Warnung liegt an
	--------------------------------------------------------------------------------
	BYTE 2: Gerätezustand/ Fehlernummer
	--------------------------------------------------------------------------------*)

(*Fehlermeldung auswerten und rangieren : Ist das Fehlerbit gesetzt, so wird die Fehlernummer ausgegeben.
  Liegt kein Fehler vor, so wird eine Null ausgegeben.*)	
 	IF stoerung 
	THEN  
		OUT_FEHLERNUMMER :=fehlernummer;
	END_IF
	
	IF NOT stoerung 
	THEN
		OUT_FEHLERNUMMER :=0;
	END_IF

//Setzten des Bits FU-Betriebbereit********************************************
	IF umrichter_bb 
	THEN 
		OUT_NICHT_BEREIT := FALSE;
		ELSE
			OUT_NICHT_BEREIT :=TRUE;
	END_IF

//Setzen des Bits FU-Störung********************************************
	IF stoerung 
		//AND NOT umrichter_bb
	THEN 
		OUT_STOERUNG := TRUE;
		ELSE 
			OUT_STOERUNG := FALSE;
	END_IF
//Setzen das Bit Warnung*************************************************
	//IF umrichter_bb
	//	 AND stoerung
	//THEN 
	//	OUT_Warnung :=TRUE;
	// 	ELSE 
	//		OUT_warnung:=FALSE;
 	//END_IF
//Ausgabe ISt-Drehzahl***************************************************
	TEMP_IST_DREHZAHL_DINT :=INT_TO_DINT(WORD_TO_INT(in_PD.PD_2_IST_DREHZAHL));
	DREHZAHL := DINT_TO_REAL(TEMP_IST_DREHZAHL_DINT);	
	
	IF IN_DREH_TAUSCH
	THEN
		OUT_DREHZAHL_IST := (DREHZAHL*0.2)*(-1);
		ELSE
			OUT_DREHZAHL_IST := DREHZAHL*0.2;
	END_IF
	

//Rechtslauf Hand-Automatik (mit Drehrichtungstausch)******************************************
	IF ((NOT IN_DREH_TAUSCH  
			AND	((IN_HAND_RECHTS AND IN_HAND)
				OR(IN_RECHTs AND NOT IN_HAND )))
 		 OR ( IN_DREH_TAUSCH
			AND((IN_HAND_LINKS AND IN_HAND)
				OR(IN_LINKS AND NOT IN_HAND ))))
	 THEN 
		rechtslauf:= TRUE;
	 	ELSE 
			rechtslauf:= FALSE;
	 END_IF

//Linkslauf Hand-Automatik (mit Drehrichtungstausch)****************************************


	IF ((NOT IN_DREH_TAUSCH  
			AND ((IN_HAND_LINKS AND IN_HAND)
				OR(IN_LINKS AND NOT IN_HAND )))
  		OR ( IN_DREH_TAUSCH
			AND ((IN_HAND_RECHTS AND IN_HAND)
					OR(IN_RECHTS AND NOT IN_HAND )))) 
  	THEN 
		linkslauf:= TRUE;
		ELSE 
			linkslauf:= FALSE;
	END_IF

//Geschwindigkeit umkopieren************************************************************
	IF IN_HAND 
	THEN 
		temp_v := IN_HAND_v;
		ELSE 
			temp_v := IN_v;
	END_IF
//Drehzahl ermitteln*************************************************************************
	temp_drehzahl_soll:= v_faktor*temp_v;

	IF temp_drehzahl_soll >= 6553.0
		THEN temp_drehzahl_soll:=6553.0;
	END_IF

	out_ist_90:=ABS(OUT_DREHZAHL_IST) >ABS((temp_drehzahl_soll/100*90));	
	out_Dreht:=ABS(OUT_DREHZAHL_IST)>1;
//Vorgabe Soll-Drehzahl***********************************************************************
	IF linkslauf
	THEN 
		out_PD.PD_2_solldrehzahl :=DWORD_TO_WORD (REAL_TO_DWORD (temp_drehzahl := ((temp_drehzahl_soll/0.2)*-1)));
		ELSE 
			 out_PD.PD_2_solldrehzahl :=DWORD_TO_WORD (REAL_TO_DWORD (temp_drehzahl := (temp_drehzahl_soll/0.2)));
	END_IF

//Vorgabe Soll-Rampe***************************************************************************
//	out_PD.PD_3_rampe :=INT_TO_WORD(IN_RAMPE);

//Reglersperre setzen**************************************************************************
	reglersperre:=IN_Reglersperre;
	freigabe_stop:=NOT IN_Reglersperre;

//Antrieb starten ,stoppen mit Rampe************************************************************
	IF rechtslauf 
		OR linkslauf
	THEN 
		freigabe_halt := TRUE;
	END_IF

//Fehler /Störung löschen*************************************************************************
	IF IN_RESET 
	THEN 
		reset:= TRUE;
		ELSE 
			reset:= FALSE;
	END_IF

//Steuerwort schreiben
	steuerbyte_1	:= BYTE_OF_BIT(
	B0:= reglersperre, 
	B1:= freigabe_stop , 
	B2:= freigabe_halt, 
	B3:= reserve_3_1, 
	B4:= reserve_4_1, 
	B5:= reserve_5_1, 
	B6:= reset, 
	B7:= reserve_7_1);
	
	steuerbyte_2 :=BYTE_OF_BIT(
	B0:= drehrichtung_motorpoti , 
	B1:= motorpoti_auf, 
	B2:= motorpoti_ab, 
	B3:= n11_n21, 
	B4:= n12_n22	 , 
	B5:= sollwert_umschaltung, 
	B6:= reserve_14  , 
	B7:= reserve_15);
    out_PD.PD_1_Steuerwort :=WORD_OF_BYTE(B1:= steuerbyte_2 , B0:=steuerbyte_1 );
	
(* Steuerwort --------------------------------------------------------------------
	BIT 0: Reglersperre
	0 = Freigabe
	1 = Regler sperren, Bremse aktivieren
	--------------------------------------------------------------------------------
	BIT 1: Freigabe/Schnellstopp
	0 = Schnellstopp
	1 = Freigabe
	--------------------------------------------------------------------------------
	BIT 2: Freigabe/Halt
	0 = Halt an Integratorrampe oder Prozess-Rampe
	1 = Freigabe
	--------------------------------------------------------------------------------
	BIT 3: Reserviert (Reservierte Bits sind generell auf Null zu setzen!)
	--------------------------------------------------------------------------------
	BIT 4: Reserviert (Reservierte Bits sind generell auf Null zu setzen!)
	--------------------------------------------------------------------------------
	BIT 5: Reserviert (Reservierte Bits sind generell auf Null zu setzen!)
	--------------------------------------------------------------------------------
	BIT 6: Reset
	0 = nicht aktiv
	0 -> 1 = anstehende Störung zurücksetzen
	--------------------------------------------------------------------------------
	BIT 7: Reserviert (Reservierte Bits sind generell auf Null zu setzen!)
	--------------------------------------------------------------------------------
	BIT 8: Drehrichtung für Motorpoti
	0 = Drehrichtung RECHTS
	1 = Drehrichtung LINKS
	--------------------------------------------------------------------------------
	BIT 10 und 9: Motorpoti Hochlauf,Motorpoti Tieflauf
	0 0 = keine Änderung
	1 0 = ab
	0 1 = auf
	1 1 = keine Änderung
	--------------------------------------------------------------------------------
	BIT 12 und 11:Anwahl der internen Festsollwerte
	n11...n13 bzw. n21...n23
	0 0 = Drehzahl-Sollwert über Prozess-Ausgangsdatenwort 2
	0 1 = interner Sollwert n11 (n21)
	1 0 = interner Sollwert n12 (n22)
	1 1 = interner Sollwert n13 (n23)
	--------------------------------------------------------------------------------
	BIT 13: Festsollwert-Umschaltung
	0 = Festsollwerte des aktivn Parametersatzes über Bit 11/12 anwählbar
	1 = Festsollwerte des anderen Parametersatzes über Bit 11/12 anwählbar
	--------------------------------------------------------------------------------
	BIT 14: Reserviert (Reservierte Bits sind generell auf Null zu setzen!)
	--------------------------------------------------------------------------------
	BIT 15: Reserviert (Reservierte Bits sind generell auf Null zu setzen!*)

END_FUNCTION_BLOCK

// ---- SRT_Allgemein/0010_Bausteine_mitDuts/POUs/FU_SEW/sub/CSV Read_Write/fb_CSVBaseRead.TcPOU
FUNCTION_BLOCK fb_CSVBaseRead
VAR_INPUT
	I_sFileName			: T_MaxString :='CSVBaseWriterTest'; (* CSV destination file path and name *)
	I_sFilePath			: T_MaxString :='\HARD DISK\Parameter\IOLINK\';
	I_sNetId				: T_AmsNetId := '5.36.121.252.1.1';	(* TwinCAT system network address *)
	I_iMaxCollumns		: INT := 10;	(*	Achtung 10 Spalten Maximal ! *)
	I_bRead				: BOOL;
	I_bReset				: BOOL;
END_VAR
VAR_OUTPUT
	Q_stCSVDatabase	: ARRAY[0..GVL_1000.MAX_CSV_BASE_ROWS] OF st_CSV_Database  ;
	Q_bError				: BOOL;
	Q_sState				: STRING;
	Q_bDone			: BOOL;
	Q_bBusy				: BOOL;
END_VAR
VAR
	bRead			: BOOL := FALSE;(* Rising edge starts program execution *)
	sNetId			: T_AmsNetId := '5.36.121.252.1.1';	(* TwinCAT system network address *)
	sFileName		:T_MaxString :='\HARD DISK\Parameter\BLDC_COEParameter.txt'; (* CSV destination file path and name *)
	sCSVLine		: T_MaxString := '';(* Single CSV text line (row, record), we are using string as record buffer (your are able to see read fields)  *)
	sCSVField		: T_MaxString := '';(* Single CSV field value (column, record field) *)
	bBusy			: BOOL;
	bError			: BOOL;
	bDone			: BOOL;
	nErrId			: UDINT;
	nRow	 		: UDINT 	:= 0;(* Row number (record) *)
	nColumn		: UDINT 	:= 0;(* Column number (record field) *)
	hFile			: UINT		:= 0;(* File handle of the source file *)
	step			: DWORD 	:= 0;
	fbFileOpen	: FB_FileOpen;(* Opens file *)
	fbFileClose	: FB_FileClose;(* Closes file *)
	fbFileGets		: FB_FileGets;(* Reads one record (line) *)
	fbReader		: FB_CSVMemBufferReader;(* Helper function block used to parse CSV data bytes (single record line) *)
	(*database		: ARRAY[0..MAX_CSV_BASE_ROWS] OF st_CSV_Database  ;*)
	(*database1		: ARRAY[0..MAX_CSV_BASE_ROWS,0..MAX_CSV_BASE_COLUMNS] OF STRING(3);*)(* Target PLC database *)
	sState			: STRING;
	Convert: BOOL ;
	i: INT;
END_VAR

(* NetID Schreiben *)
sNetId  := I_sNetId;

(* DateiNamen Schreiben *)
sFileName :=	CONCAT(I_sFilePath,I_sFileName);

(* Ablauf *)
ac_Ablauf();

(* Ausgänge *)
ac_Output();

ACTION ac_Ablauf:
bRead	:=	I_bRead;

IF NOT
I_bReset
THEN
	CASE step OF
		0:	(* Wait for rising edge at bRead variable *)
			IF bRead THEN
				bRead 	:= FALSE;
				Convert	:= FALSE;
				bBusy 		:= TRUE;
				bError		:= FALSE;
				bDone		:= FALSE;
				nErrId		:= 0;
				hFile		:= 0;
				nRow	 	:= 0;
				nColumn	:= 0;
				MEMSET( ADR( Q_stCSVDatabase ), 0, SIZEOF( Q_stCSVDatabase ) );
				step 		:= 1;
			END_IF

		1:	(* Open source file *)
			sState := 'Open source file';
			fbFileOpen(  bExecute := FALSE  );
			fbFileOpen( 	sNetId := sNetId, sPathName := sFileName, nMode := FOPEN_MODEREAD OR FOPEN_MODETEXT,(* Open file in TEXT mode! *)
							ePath := PATH_GENERIC, bExecute := TRUE );
			step := 2;
	
		2:(* Wait until open not busy *)
			sState := 'Wait until open not busy';
			fbFileOpen( bExecute := FALSE, bError => bError, nErrID => nErrID, hFile => hFile );
			IF NOT fbFileOpen.bBusy THEN
				IF NOT fbFileOpen.bError THEN
					step := 3;
				ELSE(* Error: file not found? *)
					step := 100;
				END_IF
			END_IF
	
		3:	(* Read single line (record) *)
			fbFileGets( bExecute := FALSE );
			fbFileGets( sNetId := sNetId, hFile := hFile, bExecute := TRUE );
			step := 4;
	
		4:(* Wait until read not busy *)
	
			fbFileGets( bExecute := FALSE, bError => bError, nErrID => nErrID, sLine => sCSVLine );
			IF NOT fbFileGets.bBusy THEN
				IF NOT fbFileGets.bError THEN
					IF fbFileGets.bEOF THEN
						step := 10;(* End of file reached => Close source file *)
					ELSE
	
						(* FB_FileGets returns text line without the CR (carriage return) character.
						We have to restore the CR character (replace the $L character with $R$L characters) *)
						IF RIGHT( sCSVLine, 1 ) = '$L' THEN
							sCSVLine := REPLACE( sCSVLine, '$R$L', 2, LEN( sCSVLine ) );
						END_IF
	
						step := 5;
					END_IF
				ELSE(* Error *)
					step := 100;
				END_IF
			END_IF
	
		5:(* Parse single line (record) *)
			sState := CONCAT('Reading Row -> ',UDINT_TO_STRING(nRow));
			sState := CONCAT(sState,'/ ');
			sState := CONCAT(sState,INT_TO_STRING(GVL_1000.MAX_CSV_BASE_ROWS));
	
			fbReader.eCmd := eEnumCmd_First;(* Read first field value *)
			REPEAT
				fbReader( pBuffer := ADR( sCSVLine ), cbBuffer := SIZEOF( sCSVLine ), getValue =>sCSVField );
				IF fbReader.bOk THEN
					fbReader.eCmd := eEnumCmd_Next;(* Read next field value *)
	
					IF ( nRow <= GVL_1000.MAX_CSV_BASE_ROWS ) THEN
						IF ( nColumn <= I_iMaxCollumns ) THEN
							CASE nColumn OF
								0 :	Q_stCSVDatabase[nRow].sCSV_Column1 := CSVFIELD_TO_STRING( sCSVField, FALSE );
								1:	Q_stCSVDatabase[nRow].sCSV_Column2 := CSVFIELD_TO_STRING( sCSVField, FALSE );
								2:	Q_stCSVDatabase[nRow].sCSV_Column3 := CSVFIELD_TO_STRING( sCSVField, FALSE );
								3:	Q_stCSVDatabase[nRow].sCSV_Column4 := CSVFIELD_TO_STRING( sCSVField, FALSE );
								4:	Q_stCSVDatabase[nRow].sCSV_Column5 := CSVFIELD_TO_STRING( sCSVField, FALSE );
								5:	Q_stCSVDatabase[nRow].sCSV_Column6 := CSVFIELD_TO_STRING( sCSVField, FALSE );
								6:	Q_stCSVDatabase[nRow].sCSV_Column7 := CSVFIELD_TO_STRING( sCSVField, FALSE );
								7:	Q_stCSVDatabase[nRow].sCSV_Column8 := CSVFIELD_TO_STRING( sCSVField, FALSE );
								8:	Q_stCSVDatabase[nRow].sCSV_Column9 := CSVFIELD_TO_STRING( sCSVField, FALSE );
								9:	Q_stCSVDatabase[nRow].sCSV_Column10 := CSVFIELD_TO_STRING( sCSVField, FALSE );
							END_CASE
						END_IF
					END_IF
	
					nColumn := nColumn + 1;(* Increment number of read columns *)
					IF fbReader.bCRLF THEN(* CRLF == TRUE => End of reacord reached *)
						nRow 		:= nRow + 1;(* Increment number of read records *)
						nColumn 	:= 0;(* Reset number of columns *)
					END_IF
	
				ELSE(* Error: End of record reached or all fields read *)
					step := 3;(* Try to read next line *)
				END_IF
			UNTIL NOT fbReader.bOk
			END_REPEAT
	
		10:	(* Close source file *)
			sState := 'Close source file';
			fbFileClose( bExecute := FALSE );
			fbFileClose( sNetId := sNetId, hFile := hFile, bExecute := TRUE );
			step := 11;
	
		11:(* Wait until close not busy *)
			sState := 'Wait until close not busy';
			fbFileClose( bExecute := FALSE, bError => bError, nErrID => nErrID );
			IF ( NOT fbFileClose.bBusy ) THEN
				hFile := 0;
				step := 100;
			END_IF
	
		100:	(*Convert:=TRUE;*) (* Error or ready step => cleanup *)
			Convert	:= TRUE;
			IF ( hFile <> 0 ) THEN
				step := 10; (* Close the source file *)
			ELSE
				IF NOT I_bRead
				THEN
	
					IF NOT bError
					THEN
						sState := ' Wait for start Read';
						bDone := TRUE;
					ELSE
						sState := CONCAT('Error Reading ->',UDINT_TO_STRING(nErrID));
						bDone := FALSE;
					END_IF
	
					bBusy := FALSE;
					step := 0;	(* Ready *)
	
				END_IF
			END_IF
	END_CASE
ELSE
	step 		:= 0;
	bRead 		:= FALSE;
	Convert		:= FALSE;
	bBusy 		:= FALSE;
	bError		:= FALSE;
	bDone		:= FALSE;
	nErrId		:= 0;
	hFile		:= 0;
	nRow	 	:= 0;
	nColumn		:= 0;
	MEMSET( ADR( Q_stCSVDatabase ), 0, SIZEOF( Q_stCSVDatabase ) );
END_IF
END_ACTION

ACTION ac_Output:
Q_bError	 	:=	bError;
Q_sState		:=	sState;
Q_bDone 	:=	bDone;
Q_bBusy		:=	bBusy;
END_ACTION

END_FUNCTION_BLOCK

// ---- SRT_Allgemein/0010_Bausteine_mitDuts/POUs/FU_SEW/sub/CSV Read_Write/fb_OrdnerErstellen.TcPOU
FUNCTION_BLOCK fb_OrdnerErstellen
VAR_INPUT
	I_bExecute	:BOOL;
	I_sPath		:STRING(255);	
END_VAR
VAR_OUTPUT
	Q_bDone		:BOOL;
	Q_bBusy		:BOOL;
	Q_bError	:BOOL;
	Q_iErrorID	:UDINT;	
END_VAR
VAR
	fbCreateDir	:FB_CreateDir;
END_VAR


fbCreateDir.sPathName	:=I_sPath;
fbCreateDir.bExecute		:=I_bExecute;
fbCreateDir();

Q_bBusy		:= fbCreateDir.bBusy;
Q_bError	:= fbCreateDir.bError;
Q_iErrorID	:= fbCreateDir.nErrId;

END_FUNCTION_BLOCK

// ---- SRT_Allgemein/0010_Bausteine_mitDuts/POUs/FU_SEW/sub/CSV Read_Write/fb_Parameter_CSV.TcPOU
FUNCTION_BLOCK fb_Parameter_CSV
VAR_INPUT
	I_bStartRead			:BOOL;
	I_bStartWrite			:BOOL;
	I_bReset				:BOOL;
	I_sNetId				:STRING	:=	'';
	I_sFileName			:STRING :=	'Parameter.txt';
	I_sPath				:STRING:= 	'C:\CSV\SEW';
	I_iMaxCollumns		:INT	:=4;
	I_stParameter			:ARRAY[0..GVL_1000.MAX_CSV_BASE_ROWS] OF st_MaschParameter;
END_VAR
VAR_OUTPUT
	Q_bBusy				:BOOL;
	Q_stParameter		:ARRAY[0..GVL_1000.MAX_CSV_BASE_ROWS] OF st_MaschParameter;
END_VAR
VAR
	i					:INT;
	CSV_Write			:fb_CSVBaseWrite;
	CSV_Read			:fb_CSVBaseRead;

	bCvToStrDone		:BOOL;
	bStrToCvDone		:BOOL;
	iStep: INT;

	bBusy				:BOOL;
	bErr					:BOOL;
	bDone				:BOOL;
	bWrite				:BOOL;
	bRead				:BOOL;
	sState				:STRING;
END_VAR

(*	*)
ac_Read();
(*	*)
ac_Write();
(*	*)
ac_Ablauf();

Q_bBusy:= bBusy;

ACTION ac_Ablauf:
IF I_bReset
THEN
	iStep:=0;
END_IF

CASE iStep OF

(*======================================================================================================================================*)
0:(* 	INIT *)
(*======================================================================================================================================*)
		ac_Conv_Param_To_String();
		ac_Conv_String_To_Param();

	bBusy 			:=	FALSE;
	bWrite			:=	FALSE;
	bRead			:=	FALSE;

	IF 	I_bStartWrite
	THEN
		iStep := iStep +10;
	END_IF

	IF 	I_bStartRead
	THEN
		iStep := iStep +100;
	END_IF

(*======================================================================================================================================*)
10:(* 	INIT *)
(*======================================================================================================================================*)
		ac_Conv_Param_To_String();

	sState			:=	'WRITE-INIT';
	bDone			:=	FALSE;
	bErr				:=	FALSE;
	bBusy 			:= 	TRUE;
	bCvToStrDone	:= 	FALSE;

	iStep 			:= 	iStep +10;

(*======================================================================================================================================*)
20:(* 	Konvertierung  *)
(*======================================================================================================================================*)
	sState			:=	'WRITE-CONVERT';

		ac_Conv_Param_To_String();

	IF	bCvToStrDone
	THEN
		iStep 			:= 	iStep +10;
	END_IF

(*======================================================================================================================================*)
30:(* 	Write *)
(*======================================================================================================================================*)
	sState			:=	'WRITE-START';
	bWrite			:=	TRUE;

	IF CSV_Write.bBusy
		AND NOT CSV_Write.bError
	THEN
		iStep		:=	iStep+10;
	ELSIF
		CSV_Write.Q_bError
	THEN
		iStep		:=	-20;
	END_IF

(*======================================================================================================================================*)
40:(* 	Warte auf Fertig *)
(*======================================================================================================================================*)
	sState			:=	'WRITE-START';
	bWrite			:=	FALSE;

	IF	NOT CSV_Write.bBusy
		AND CSV_Write.Q_bDone
		AND NOT CSV_Write.bError
	THEN
		bDone			:=	TRUE;
	END_IF

	IF NOT CSV_Write.bBusy
		AND CSV_Write.Q_bDone
		AND NOT I_bStartWrite
	THEN
		sState		:=	'WRITE-DONE';
		iStep		:=	0;
	ELSIF
		CSV_Write.Q_bError
	THEN
		iStep		:=	-20;
	END_IF


(*======================================================================================================================================*)
100:(* 	INIT *)
(*======================================================================================================================================*)
		ac_Conv_Param_To_String();

	sState			:=	'READ-INIT';
	bDone			:=	FALSE;
	bErr				:=	FALSE;
	bBusy 			:= 	TRUE;
	bStrToCvDone	:= 	FALSE;

	iStep 			:= 	iStep +20;

(*======================================================================================================================================*)
120:(* 	READ  *)
(*======================================================================================================================================*)
	sState			:=	'READ-START';
	bRead			:=	TRUE;

	IF CSV_Read.bBusy
		AND NOT CSV_Read.bError
	THEN
		iStep		:=	iStep+10;
	ELSIF
		CSV_Read.Q_bError
	THEN
		iStep		:=	-130;
	END_IF

(*======================================================================================================================================*)
130:(* 	READ *)
(*======================================================================================================================================*)
	sState			:=	'READ-WAIT-DONE';
	bRead			:=	FALSE;

	IF NOT CSV_Read.bBusy
		AND CSV_Read.Q_bDone
	THEN
		iStep		:=	iStep+10;
	ELSIF
		CSV_Read.Q_bError
	THEN
		iStep		:=	-130;
	END_IF

(*======================================================================================================================================*)
140:(* 	Konvertierung in Parameter  *)
(*======================================================================================================================================*)
	sState			:=	'READ-CONVERT';

		ac_Conv_String_To_Param();

	IF	bStrToCvDone
	THEN
		bDone			:=	TRUE;
	END_IF

	IF	bStrToCvDone
		AND NOT I_bStartRead
	THEN
		sState			:=	'READ-DONE';
		iStep 			:= 	0;
	END_IF

(*======================================================================================================================================*)
(* 	ERRORs  *)
(*======================================================================================================================================*)

-20:
	sState 		:=	CONCAT('CSV-WRITE-ERROR: ',CSV_Write.Q_sState);
	bErr 		:= 	TRUE;
	iStep 		:= 	-999;

-130:
	sState 		:=	CONCAT('CSV-READ-ERROR: ',CSV_Read.Q_sState);
	bErr 		:= 	TRUE;
	iStep 		:= 	-999;

-999:
	IF  NOT I_bStartRead
	THEN
		iStep 			:= 	0;
	END_IF

END_CASE
END_ACTION

ACTION ac_Conv_Param_To_String:
FOR i := 0 TO GVL_1000.MAX_CSV_BASE_ROWS BY 1 DO
	CSV_Write.I_stCSVDatabase[i].sCSV_Column1	:=	I_stParameter[i].sName;
	CSV_Write.I_stCSVDatabase[i].sCSV_Column2	:=	LREAL_TO_STRING(I_stParameter[i].nWert);
	CSV_Write.I_stCSVDatabase[i].sCSV_Column3	:=	BOOL_TO_STRING(I_stParameter[i].bWert);
	CSV_Write.I_stCSVDatabase[i].sCSV_Column4	:=	LREAL_TO_STRING(TIME_TO_LREAL(I_stParameter[i].tWert));

	IF i >= GVL_1000.MAX_CSV_BASE_ROWS
	THEN
		bCvToStrDone	:= 	TRUE;
	ELSE
		bCvToStrDone	:=	FALSE;
	END_IF

END_FOR
END_ACTION

ACTION ac_Conv_String_To_Param:
;
FOR i := 0 TO GVL_1000.MAX_CSV_BASE_ROWS BY 1 DO

	Q_stParameter[i].sName			:=		CSV_Read.Q_stCSVDatabase[i].sCSV_Column1;
	Q_stParameter[i].nWert				:=		STRING_TO_LREAL(CSV_Read.Q_stCSVDatabase[i].sCSV_Column2);
	Q_stParameter[i].bWert				:=		STRING_TO_BOOL(CSV_Read.Q_stCSVDatabase[i].sCSV_Column3);
	Q_stParameter[i].tWert				:=		LREAL_TO_TIME(STRING_TO_LREAL(CSV_Read.Q_stCSVDatabase[i].sCSV_Column4));

	IF i >= GVL_1000.MAX_CSV_BASE_ROWS
	THEN
		bStrToCvDone	:= 	TRUE;
	ELSE
		bStrToCvDone	:=	FALSE;
	END_IF

END_FOR
END_ACTION

ACTION ac_Read:
CSV_Read(
	I_sFileName:= 		I_sFileName,
	I_sFilePath:= 			I_sPath,
	I_sNetId:= 			I_sNetId,
	I_iMaxCollumns:= 		I_iMaxCollumns,
	I_bRead:=			bRead ,
	I_bReset:= 			I_bReset,
	Q_stCSVDatabase=> ,
	Q_bError=> ,
	Q_sState=> ,
	Q_bDone=> , 
	Q_bBusy=> );
END_ACTION

ACTION ac_Write:
CSV_Write(
	I_sFileName:= 		I_sFileName,
	I_sFilePath:= 			I_sPath,
	I_sNetId:= 			I_sNetId,
	I_stCSVDatabase:=	 ,
	I_iMaxCollumns:= 		I_iMaxCollumns,
	I_bWrite:= 			bWrite,
	I_bReset:= ,
	I_sTimeStamp:= , 
	Q_bError=> , 
	Q_sState=> , 
	Q_bDone=> , 
	Q_bBusy=> );
END_ACTION

END_FUNCTION_BLOCK

// ---- SRT_Allgemein/0010_Bausteine_mitDuts/POUs/Safety/FB_InfoConnection_1918.TcPOU
FUNCTION_BLOCK FB_InfoConnection_1918
VAR_INPUT
	stInfoData: ST_InfoDataConnection_1918;
	eMode: E_ModeLanguage := 1;
END_VAR
VAR_OUTPUT
	sState: STRING;
	sDiag: STRING;
	bChannel1: BOOL;
	bChannel2: BOOL;
	bChannel3: BOOL;
	bChannel4: BOOL;
	bChannel5: BOOL;
	bChannel6: BOOL;
	bChannel7: BOOL;
	bChannel8: BOOL;
END_VAR
VAR
	arTextState: ARRAY[1..2] OF STRING;
	arTextDiag: ARRAY[1..2] OF STRING;
END_VAR

